(* IEC 61131-3 sources: elnaProjects/ElpcLogic/PomarKc7Changed/FunctionBlocks (part 5) *)

(* ---- OPC_AI_SET.st ---- *)
FUNCTION_BLOCK OPC_AI_SET

VAR_EXTERNAL
	ai : aiConfig;
	AI_Tstali_statora_kanal_1_HL : LREAL;
	AI_Tstali_statora_kanal_1_LL : LREAL;
	AI_Tstali_statora_kanal_1_command : UINT;
	AI_Tstali_statora_kanal_1_newHL : LREAL;
	AI_Tstali_statora_kanal_1_newLL : LREAL;
	AI_Tstali_statora_kanal_1_status : UDINT;
	AI_Tstali_statora_kanal_1_value : LREAL;
	AI_Tstali_statora_kanal_1_HW : LREAL;
	AI_Tstali_statora_kanal_1_newHW : LREAL;
	AI_Tstali_statora_kanal_2_HL : LREAL;
	AI_Tstali_statora_kanal_2_LL : LREAL;
	AI_Tstali_statora_kanal_2_command : UINT;
	AI_Tstali_statora_kanal_2_newHL : LREAL;
	AI_Tstali_statora_kanal_2_newLL : LREAL;
	AI_Tstali_statora_kanal_2_status : UDINT;
	AI_Tstali_statora_kanal_2_value : LREAL;
	AI_Tstali_statora_kanal_2_HW : LREAL;
	AI_Tstali_statora_kanal_2_newHW : LREAL;
	AI_Tstali_statora_kanal_3_HL : LREAL;
	AI_Tstali_statora_kanal_3_LL : LREAL;
	AI_Tstali_statora_kanal_3_command : UINT;
	AI_Tstali_statora_kanal_3_newHL : LREAL;
	AI_Tstali_statora_kanal_3_newLL : LREAL;
	AI_Tstali_statora_kanal_3_status : UDINT;
	AI_Tstali_statora_kanal_3_value : LREAL;
	AI_Tstali_statora_kanal_3_HW : LREAL;
	AI_Tstali_statora_kanal_3_newHW : LREAL;
	AI_Tmedi_statora_kanal_1_HL : LREAL;
	AI_Tmedi_statora_kanal_1_LL : LREAL;
	AI_Tmedi_statora_kanal_1_command : UINT;
	AI_Tmedi_statora_kanal_1_newHL : LREAL;
	AI_Tmedi_statora_kanal_1_newLL : LREAL;
	AI_Tmedi_statora_kanal_1_status : UDINT;
	AI_Tmedi_statora_kanal_1_value : LREAL;
	AI_Tmedi_statora_kanal_1_HW : LREAL;
	AI_Tmedi_statora_kanal_1_newHW : LREAL;
	AI_Tmedi_statora_kanal_2_HL : LREAL;
	AI_Tmedi_statora_kanal_2_LL : LREAL;
	AI_Tmedi_statora_kanal_2_command : UINT;
	AI_Tmedi_statora_kanal_2_newHL : LREAL;
	AI_Tmedi_statora_kanal_2_newLL : LREAL;
	AI_Tmedi_statora_kanal_2_status : UDINT;
	AI_Tmedi_statora_kanal_2_value : LREAL;
	AI_Tmedi_statora_kanal_2_HW : LREAL;
	AI_Tmedi_statora_kanal_2_newHW : LREAL;
	AI_Tmedi_statora_kanal_3_HL : LREAL;
	AI_Tmedi_statora_kanal_3_LL : LREAL;
	AI_Tmedi_statora_kanal_3_command : UINT;
	AI_Tmedi_statora_kanal_3_newHL : LREAL;
	AI_Tmedi_statora_kanal_3_newLL : LREAL;
	AI_Tmedi_statora_kanal_3_status : UDINT;
	AI_Tmedi_statora_kanal_3_value : LREAL;
	AI_Tmedi_statora_kanal_3_HW : LREAL;
	AI_Tmedi_statora_kanal_3_newHW : LREAL;
	AI_Toporno_podshipnika_EDT_1_HL : LREAL;
	AI_Toporno_podshipnika_EDT_1_LL : LREAL;
	AI_Toporno_podshipnika_EDT_1_command : UINT;
	AI_Toporno_podshipnika_EDT_1_newHL : LREAL;
	AI_Toporno_podshipnika_EDT_1_newLL : LREAL;
	AI_Toporno_podshipnika_EDT_1_status : UDINT;
	AI_Toporno_podshipnika_EDT_1_value : LREAL;
	AI_Toporno_podshipnika_EDT_1_HW : LREAL;
	AI_Toporno_podshipnika_EDT_1_newHW : LREAL;
	AI_Toporno_podshipnika_EDT_1_HA : LREAL;
	AI_Toporno_podshipnika_EDT_1_newHA : LREAL;
	AI_Toy_podshipnika_EDT_2_HL : LREAL;
	AI_Toy_podshipnika_EDT_2_LL : LREAL;
	AI_Toy_podshipnika_EDT_2_command : UINT;
	AI_Toy_podshipnika_EDT_2_newHL : LREAL;
	AI_Toy_podshipnika_EDT_2_newLL : LREAL;
	AI_Toy_podshipnika_EDT_2_status : UDINT;
	AI_Toy_podshipnika_EDT_2_value : LREAL;
	AI_Toy_podshipnika_EDT_2_HW : LREAL;
	AI_Toy_podshipnika_EDT_2_newHW : LREAL;
	AI_Toy_podshipnika_EDT_2_HA : LREAL;
	AI_Toy_podshipnika_EDT_2_newHA : LREAL;
	AI_Toy_podshipnika_kol_EDT_3_HL : LREAL;
	AI_Toy_podshipnika_kol_EDT_3_LL : LREAL;
	AI_Toy_podshipnika_kol_EDT_3_command : UINT;
	AI_Toy_podshipnika_kol_EDT_3_newHL : LREAL;
	AI_Toy_podshipnika_kol_EDT_3_newLL : LREAL;
	AI_Toy_podshipnika_kol_EDT_3_status : UDINT;
	AI_Toy_podshipnika_kol_EDT_3_value : LREAL;
	AI_Toy_podshipnika_kol_EDT_3_HW : LREAL;
	AI_Toy_podshipnika_kol_EDT_3_newHW : LREAL;
	AI_Toy_podshipnika_kol_EDT_3_HA : LREAL;
	AI_Toy_podshipnika_kol_EDT_3_newHA : LREAL;
	AI_Toy_podshipnika_kol_EDT_4_HL : LREAL;
	AI_Toy_podshipnika_kol_EDT_4_LL : LREAL;
	AI_Toy_podshipnika_kol_EDT_4_command : UINT;
	AI_Toy_podshipnika_kol_EDT_4_newHL : LREAL;
	AI_Toy_podshipnika_kol_EDT_4_newLL : LREAL;
	AI_Toy_podshipnika_kol_EDT_4_status : UDINT;
	AI_Toy_podshipnika_kol_EDT_4_value : LREAL;
	AI_Toy_podshipnika_kol_EDT_4_HW : LREAL;
	AI_Toy_podshipnika_kol_EDT_4_newHW : LREAL;
	AI_Toy_podshipnika_kol_EDT_4_HA : LREAL;
	AI_Toy_podshipnika_kol_EDT_4_newHA : LREAL;
	AI_Toy_podshipnika_shest_red_EDT_5_HL : LREAL;
	AI_Toy_podshipnika_shest_red_EDT_5_LL : LREAL;
	AI_Toy_podshipnika_shest_red_EDT_5_command : UINT;
	AI_Toy_podshipnika_shest_red_EDT_5_newHL : LREAL;
	AI_Toy_podshipnika_shest_red_EDT_5_newLL : LREAL;
	AI_Toy_podshipnika_shest_red_EDT_5_status : UDINT;
	AI_Toy_podshipnika_shest_red_EDT_5_value : LREAL;
	AI_Toy_podshipnika_shest_red_EDT_5_HW : LREAL;
	AI_Toy_podshipnika_shest_red_EDT_5_newHW : LREAL;
	AI_Toy_podshipnika_shest_red_EDT_5_HA : LREAL;
	AI_Toy_podshipnika_shest_red_EDT_5_newHA : LREAL;
	AI_Ty_podshipnika_red_EDT_6_HL : LREAL;
	AI_Ty_podshipnika_red_EDT_6_LL : LREAL;
	AI_Ty_podshipnika_red_EDT_6_command : UINT;
	AI_Ty_podshipnika_red_EDT_6_newHL : LREAL;
	AI_Ty_podshipnika_red_EDT_6_newLL : LREAL;
	AI_Ty_podshipnika_red_EDT_6_status : UDINT;
	AI_Ty_podshipnika_red_EDT_6_value : LREAL;
	AI_Ty_podshipnika_red_EDT_6_HW : LREAL;
	AI_Ty_podshipnika_red_EDT_6_newHW : LREAL;
	AI_Ty_podshipnika_red_EDT_6_HA : LREAL;
	AI_Ty_podshipnika_red_EDT_6_newHA : LREAL;
	AI_Ty_podshipnika_nagnet_EDT_7_1_HL : LREAL;
	AI_Ty_podshipnika_nagnet_EDT_7_1_LL : LREAL;
	AI_Ty_podshipnika_nagnet_EDT_7_1_command : UINT;
	AI_Ty_podshipnika_nagnet_EDT_7_1_newHL : LREAL;
	AI_Ty_podshipnika_nagnet_EDT_7_1_newLL : LREAL;
	AI_Ty_podshipnika_nagnet_EDT_7_1_status : UDINT;
	AI_Ty_podshipnika_nagnet_EDT_7_1_value : LREAL;
	AI_Ty_podshipnika_nagnet_EDT_7_1_HW : LREAL;
	AI_Ty_podshipnika_nagnet_EDT_7_1_newHW : LREAL;
	AI_Ty_podshipnika_nagnet_EDT_7_1_HA : LREAL;
	AI_Ty_podshipnika_nagnet_EDT_7_1_newHA : LREAL;
	AI_Ty_podshipnika_nagnet_EDT_7_2_HL : LREAL;
	AI_Ty_podshipnika_nagnet_EDT_7_2_LL : LREAL;
	AI_Ty_podshipnika_nagnet_EDT_7_2_command : UINT;
	AI_Ty_podshipnika_nagnet_EDT_7_2_newHL : LREAL;
	AI_Ty_podshipnika_nagnet_EDT_7_2_newLL : LREAL;
	AI_Ty_podshipnika_nagnet_EDT_7_2_status : UDINT;
	AI_Ty_podshipnika_nagnet_EDT_7_2_value : LREAL;
	AI_Ty_podshipnika_nagnet_EDT_7_2_HW : LREAL;
	AI_Ty_podshipnika_nagnet_EDT_7_2_newHW : LREAL;
	AI_Ty_podshipnika_nagnet_EDT_7_2_HA : LREAL;
	AI_Ty_podshipnika_nagnet_EDT_7_2_newHA : LREAL;
	AI_Toy_podshipnika_svobod_konca_EDT_8_1_HL : LREAL;
	AI_Toy_podshipnika_svobod_konca_EDT_8_1_LL : LREAL;
	AI_Toy_podshipnika_svobod_konca_EDT_8_1_command : UINT;
	AI_Toy_podshipnika_svobod_konca_EDT_8_1_newHL : LREAL;
	AI_Toy_podshipnika_svobod_konca_EDT_8_1_newLL : LREAL;
	AI_Toy_podshipnika_svobod_konca_EDT_8_1_status : UDINT;
	AI_Toy_podshipnika_svobod_konca_EDT_8_1_value : LREAL;
	AI_Toy_podshipnika_svobod_konca_EDT_8_1_HW : LREAL;
	AI_Toy_podshipnika_svobod_konca_EDT_8_1_newHW : LREAL;
	AI_Toy_podshipnika_svobod_konca_EDT_8_1_HA : LREAL;
	AI_Toy_podshipnika_svobod_konca_EDT_8_1_newHA : LREAL;
	AI_Toy_podshipnika_svobod_konca_EDT_8_2_HL : LREAL;
	AI_Toy_podshipnika_svobod_konca_EDT_8_2_LL : LREAL;
	AI_Toy_podshipnika_svobod_konca_EDT_8_2_command : UINT;
	AI_Toy_podshipnika_svobod_konca_EDT_8_2_newHL : LREAL;
	AI_Toy_podshipnika_svobod_konca_EDT_8_2_newLL : LREAL;
	AI_Toy_podshipnika_svobod_konca_EDT_8_2_status : UDINT;
	AI_Toy_podshipnika_svobod_konca_EDT_8_2_value : LREAL;
	AI_Toy_podshipnika_svobod_konca_EDT_8_2_HW : LREAL;
	AI_Toy_podshipnika_svobod_konca_EDT_8_2_newHW : LREAL;
	AI_Toy_podshipnika_svobod_konca_EDT_8_2_HA : LREAL;
	AI_Toy_podshipnika_svobod_konca_EDT_8_2_newHA : LREAL;
	AI_Toy_podshipnika_rab_kol_EDT_9_1_HL : LREAL;
	AI_Toy_podshipnika_rab_kol_EDT_9_1_LL : LREAL;
	AI_Toy_podshipnika_rab_kol_EDT_9_1_command : UINT;
	AI_Toy_podshipnika_rab_kol_EDT_9_1_newHL : LREAL;
	AI_Toy_podshipnika_rab_kol_EDT_9_1_newLL : LREAL;
	AI_Toy_podshipnika_rab_kol_EDT_9_1_status : UDINT;
	AI_Toy_podshipnika_rab_kol_EDT_9_1_value : LREAL;
	AI_Toy_podshipnika_rab_kol_EDT_9_1_HW : LREAL;
	AI_Toy_podshipnika_rab_kol_EDT_9_1_newHW : LREAL;
	AI_Toy_podshipnika_rab_kol_EDT_9_1_HA : LREAL;
	AI_Toy_podshipnika_rab_kol_EDT_9_1_newHA : LREAL;
	AI_Toy_podshipnika_rab_kol_EDT_9_2_HL : LREAL;
	AI_Toy_podshipnika_rab_kol_EDT_9_2_LL : LREAL;
	AI_Toy_podshipnika_rab_kol_EDT_9_2_command : UINT;
	AI_Toy_podshipnika_rab_kol_EDT_9_2_newHL : LREAL;
	AI_Toy_podshipnika_rab_kol_EDT_9_2_newLL : LREAL;
	AI_Toy_podshipnika_rab_kol_EDT_9_2_status : UDINT;
	AI_Toy_podshipnika_rab_kol_EDT_9_2_value : LREAL;
	AI_Toy_podshipnika_rab_kol_EDT_9_2_HW : LREAL;
	AI_Toy_podshipnika_rab_kol_EDT_9_2_newHW : LREAL;
	AI_Toy_podshipnika_rab_kol_EDT_9_2_HA : LREAL;
	AI_Toy_podshipnika_rab_kol_EDT_9_2_newHA : LREAL;
	AI_Toy_podshipnika_nerab_kol_EDT_10_1_HL : LREAL;
	AI_Toy_podshipnika_nerab_kol_EDT_10_1_LL : LREAL;
	AI_Toy_podshipnika_nerab_kol_EDT_10_1_command : UINT;
	AI_Toy_podshipnika_nerab_kol_EDT_10_1_newHL : LREAL;
	AI_Toy_podshipnika_nerab_kol_EDT_10_1_newLL : LREAL;
	AI_Toy_podshipnika_nerab_kol_EDT_10_1_status : UDINT;
	AI_Toy_podshipnika_nerab_kol_EDT_10_1_value : LREAL;
	AI_Toy_podshipnika_nerab_kol_EDT_10_1_HW : LREAL;
	AI_Toy_podshipnika_nerab_kol_EDT_10_1_newHW : LREAL;
	AI_Toy_podshipnika_nerab_kol_EDT_10_1_HA : LREAL;
	AI_Toy_podshipnika_nerab_kol_EDT_10_1_newHA : LREAL;
	AI_Toy_podshipnika_nerab_kol_EDT_10_2_HL : LREAL;
	AI_Toy_podshipnika_nerab_kol_EDT_10_2_LL : LREAL;
	AI_Toy_podshipnika_nerab_kol_EDT_10_2_command : UINT;
	AI_Toy_podshipnika_nerab_kol_EDT_10_2_newHL : LREAL;
	AI_Toy_podshipnika_nerab_kol_EDT_10_2_newLL : LREAL;
	AI_Toy_podshipnika_nerab_kol_EDT_10_2_status : UDINT;
	AI_Toy_podshipnika_nerab_kol_EDT_10_2_value : LREAL;
	AI_Toy_podshipnika_nerab_kol_EDT_10_2_HW : LREAL;
	AI_Toy_podshipnika_nerab_kol_EDT_10_2_newHW : LREAL;
	AI_Toy_podshipnika_nerab_kol_EDT_10_2_HA : LREAL;
	AI_Toy_podshipnika_nerab_kol_EDT_10_2_newHA : LREAL;
	AI_Tholodnogo_vozduha_ED_kanal_1_HL : LREAL;
	AI_Tholodnogo_vozduha_ED_kanal_1_LL : LREAL;
	AI_Tholodnogo_vozduha_ED_kanal_1_command : UINT;
	AI_Tholodnogo_vozduha_ED_kanal_1_newHL : LREAL;
	AI_Tholodnogo_vozduha_ED_kanal_1_newLL : LREAL;
	AI_Tholodnogo_vozduha_ED_kanal_1_status : UDINT;
	AI_Tholodnogo_vozduha_ED_kanal_1_value : LREAL;
	AI_Tholodnogo_vozduha_ED_kanal_1_HW : LREAL;
	AI_Tholodnogo_vozduha_ED_kanal_1_newHW : LREAL;
	AI_Tholodnogo_vozduha_ED_kanal_2_HL : LREAL;
	AI_Tholodnogo_vozduha_ED_kanal_2_LL : LREAL;
	AI_Tholodnogo_vozduha_ED_kanal_2_command : UINT;
	AI_Tholodnogo_vozduha_ED_kanal_2_newHL : LREAL;
	AI_Tholodnogo_vozduha_ED_kanal_2_newLL : LREAL;
	AI_Tholodnogo_vozduha_ED_kanal_2_status : UDINT;
	AI_Tholodnogo_vozduha_ED_kanal_2_value : LREAL;
	AI_Tholodnogo_vozduha_ED_kanal_2_HW : LREAL;
	AI_Tholodnogo_vozduha_ED_kanal_2_newHW : LREAL;
	AI_Tgorjachego_vozduha_ED_kanal_1_HL : LREAL;
	AI_Tgorjachego_vozduha_ED_kanal_1_LL : LREAL;
	AI_Tgorjachego_vozduha_ED_kanal_1_command : UINT;
	AI_Tgorjachego_vozduha_ED_kanal_1_newHL : LREAL;
	AI_Tgorjachego_vozduha_ED_kanal_1_newLL : LREAL;
	AI_Tgorjachego_vozduha_ED_kanal_1_status : UDINT;
	AI_Tgorjachego_vozduha_ED_kanal_1_value : LREAL;
	AI_Tgorjachego_vozduha_ED_kanal_1_HW : LREAL;
	AI_Tgorjachego_vozduha_ED_kanal_1_newHW : LREAL;
	AI_Tgorjachego_vozduha_ED_kanal_2_HL : LREAL;
	AI_Tgorjachego_vozduha_ED_kanal_2_LL : LREAL;
	AI_Tgorjachego_vozduha_ED_kanal_2_command : UINT;
	AI_Tgorjachego_vozduha_ED_kanal_2_newHL : LREAL;
	AI_Tgorjachego_vozduha_ED_kanal_2_newLL : LREAL;
	AI_Tgorjachego_vozduha_ED_kanal_2_status : UDINT;
	AI_Tgorjachego_vozduha_ED_kanal_2_value : LREAL;
	AI_Tgorjachego_vozduha_ED_kanal_2_HW : LREAL;
	AI_Tgorjachego_vozduha_ED_kanal_2_newHW : LREAL;
	AI_Tnarujnogo_vozduha_HL : LREAL;
	AI_Tnarujnogo_vozduha_LL : LREAL;
	AI_Tnarujnogo_vozduha_command : UINT;
	AI_Tnarujnogo_vozduha_newHL : LREAL;
	AI_Tnarujnogo_vozduha_newLL : LREAL;
	AI_Tnarujnogo_vozduha_status : UDINT;
	AI_Tnarujnogo_vozduha_value : LREAL;
	AI_Tnarujnogo_vozduha_HW : LREAL;
	AI_Tnarujnogo_vozduha_newHW : LREAL;
	AI_Tgaza_na_vhode_H_HL : LREAL;
	AI_Tgaza_na_vhode_H_LL : LREAL;
	AI_Tgaza_na_vhode_H_command : UINT;
	AI_Tgaza_na_vhode_H_newHL : LREAL;
	AI_Tgaza_na_vhode_H_newLL : LREAL;
	AI_Tgaza_na_vhode_H_status : UDINT;
	AI_Tgaza_na_vhode_H_value : LREAL;
	AI_Tgaza_na_vhode_H_HW : LREAL;
	AI_Tgaza_na_vhode_H_newHW : LREAL;
	AI_Tgaza_na_vyhode_H_HL : LREAL;
	AI_Tgaza_na_vyhode_H_LL : LREAL;
	AI_Tgaza_na_vyhode_H_command : UINT;
	AI_Tgaza_na_vyhode_H_newHL : LREAL;
	AI_Tgaza_na_vyhode_H_newLL : LREAL;
	AI_Tgaza_na_vyhode_H_status : UDINT;
	AI_Tgaza_na_vyhode_H_value : LREAL;
	AI_Tgaza_na_vyhode_H_HW : LREAL;
	AI_Tgaza_na_vyhode_H_newHW : LREAL;
	AI_Tgaza_na_vyhode_H_HA : LREAL;
	AI_Tgaza_na_vyhode_H_newHA : LREAL;
	AI_Tmasla_do_AVOM_HL : LREAL;
	AI_Tmasla_do_AVOM_LL : LREAL;
	AI_Tmasla_do_AVOM_command : UINT;
	AI_Tmasla_do_AVOM_newHL : LREAL;
	AI_Tmasla_do_AVOM_newLL : LREAL;
	AI_Tmasla_do_AVOM_status : UDINT;
	AI_Tmasla_do_AVOM_value : LREAL;
	AI_Tmasla_do_AVOM_HW : LREAL;
	AI_Tmasla_do_AVOM_newHW : LREAL;
	AI_Tmasla_posle_AVOM_HL : LREAL;
	AI_Tmasla_posle_AVOM_LL : LREAL;
	AI_Tmasla_posle_AVOM_command : UINT;
	AI_Tmasla_posle_AVOM_newHL : LREAL;
	AI_Tmasla_posle_AVOM_newLL : LREAL;
	AI_Tmasla_posle_AVOM_status : UDINT;
	AI_Tmasla_posle_AVOM_value : LREAL;
	AI_Tmasla_posle_AVOM_HW : LREAL;
	AI_Tmasla_posle_AVOM_newHW : LREAL;
	AI_Tmasla_MB_HL : LREAL;
	AI_Tmasla_MB_LL : LREAL;
	AI_Tmasla_MB_command : UINT;
	AI_Tmasla_MB_newHL : LREAL;
	AI_Tmasla_MB_newLL : LREAL;
	AI_Tmasla_MB_status : UDINT;
	AI_Tmasla_MB_value : LREAL;
	AI_Tmasla_MB_HW : LREAL;
	AI_Tmasla_MB_newHW : LREAL;
	AI_Tmasla_MB_TEN_HL : LREAL;
	AI_Tmasla_MB_TEN_LL : LREAL;
	AI_Tmasla_MB_TEN_command : UINT;
	AI_Tmasla_MB_TEN_newHL : LREAL;
	AI_Tmasla_MB_TEN_newLL : LREAL;
	AI_Tmasla_MB_TEN_status : UDINT;
	AI_Tmasla_MB_TEN_value : LREAL;
	AI_Tmasla_MB_TEN_HW : LREAL;
	AI_Tmasla_MB_TEN_newHW : LREAL;
	AI_Tshu_HL : LREAL;
	AI_Tshu_LL : LREAL;
	AI_Tshu_command : UINT;
	AI_Tshu_newHL : LREAL;
	AI_Tshu_newLL : LREAL;
	AI_Tshu_status : UDINT;
	AI_Tshu_value : LREAL;
	AI_Pmaslo_sm_nizkoe_HL : LREAL;
	AI_Pmaslo_sm_nizkoe_LL : LREAL;
	AI_Pmaslo_sm_nizkoe_command : UINT;
	AI_Pmaslo_sm_nizkoe_newHL : LREAL;
	AI_Pmaslo_sm_nizkoe_newLL : LREAL;
	AI_Pmaslo_sm_nizkoe_status : UDINT;
	AI_Pmaslo_sm_nizkoe_value : LREAL;
	AI_Pmaslo_sm_nizkoe_LW : LREAL;
	AI_Pmaslo_sm_nizkoe_newLW : LREAL;
	AI_Pmaslo_sm_nizkoe_LA : LREAL;
	AI_Pmaslo_sm_nizkoe_newLA : LREAL;
	AI_Pmaslo_sm_vysokoe_HL : LREAL;
	AI_Pmaslo_sm_vysokoe_LL : LREAL;
	AI_Pmaslo_sm_vysokoe_command : UINT;
	AI_Pmaslo_sm_vysokoe_newHL : LREAL;
	AI_Pmaslo_sm_vysokoe_newLL : LREAL;
	AI_Pmaslo_sm_vysokoe_status : UDINT;
	AI_Pmaslo_sm_vysokoe_value : LREAL;
	AI_Pmaslo_sm_vysokoe_LW : LREAL;
	AI_Pmaslo_sm_vysokoe_newLW : LREAL;
	AI_Pmaslo_sm_vysokoe_LA : LREAL;
	AI_Pmaslo_sm_vysokoe_newLA : LREAL;
	AI_Pmasla_posle_GNS_HL : LREAL;
	AI_Pmasla_posle_GNS_LL : LREAL;
	AI_Pmasla_posle_GNS_command : UINT;
	AI_Pmasla_posle_GNS_newHL : LREAL;
	AI_Pmasla_posle_GNS_newLL : LREAL;
	AI_Pmasla_posle_GNS_status : UDINT;
	AI_Pmasla_posle_GNS_value : LREAL;
	AI_Pmasla_posle_GNS_HW : LREAL;
	AI_Pmasla_posle_GNS_newHW : LREAL;
	AI_Pmasla_posle_GNS_LW : LREAL;
	AI_Pmasla_posle_GNS_newLW : LREAL;
	AI_Pmasla_posle_NU_HL : LREAL;
	AI_Pmasla_posle_NU_LL : LREAL;
	AI_Pmasla_posle_NU_command : UINT;
	AI_Pmasla_posle_NU_newHL : LREAL;
	AI_Pmasla_posle_NU_newLL : LREAL;
	AI_Pmasla_posle_NU_status : UDINT;
	AI_Pmasla_posle_NU_value : LREAL;
	AI_Pmasla_posle_NU_LW : LREAL;
	AI_Pmasla_posle_NU_newLW : LREAL;
	AI_Pgaza_na_vhode_nagnetatelia_HL : LREAL;
	AI_Pgaza_na_vhode_nagnetatelia_LL : LREAL;
	AI_Pgaza_na_vhode_nagnetatelia_command : UINT;
	AI_Pgaza_na_vhode_nagnetatelia_newHL : LREAL;
	AI_Pgaza_na_vhode_nagnetatelia_newLL : LREAL;
	AI_Pgaza_na_vhode_nagnetatelia_status : UDINT;
	AI_Pgaza_na_vhode_nagnetatelia_value : LREAL;
	AI_Pgaza_na_vhode_nagnetatelia_LW : LREAL;
	AI_Pgaza_na_vhode_nagnetatelia_newLW : LREAL;
	AI_Pgaza_na_vyhode_nagnetatelia_HL : LREAL;
	AI_Pgaza_na_vyhode_nagnetatelia_LL : LREAL;
	AI_Pgaza_na_vyhode_nagnetatelia_command : UINT;
	AI_Pgaza_na_vyhode_nagnetatelia_newHL : LREAL;
	AI_Pgaza_na_vyhode_nagnetatelia_newLL : LREAL;
	AI_Pgaza_na_vyhode_nagnetatelia_status : UDINT;
	AI_Pgaza_na_vyhode_nagnetatelia_value : LREAL;
	AI_Pgaza_na_vyhode_nagnetatelia_LW : LREAL;
	AI_Pgaza_na_vyhode_nagnetatelia_newLW : LREAL;
	AI_Pgaza_na_vyhode_nagnetatelia_HA : LREAL;
	AI_Pgaza_na_vyhode_nagnetatelia_newHA : LREAL;
	AI_Pimpuls_gaz_HL : LREAL;
	AI_Pimpuls_gaz_LL : LREAL;
	AI_Pimpuls_gaz_command : UINT;
	AI_Pimpuls_gaz_newHL : LREAL;
	AI_Pimpuls_gaz_newLL : LREAL;
	AI_Pimpuls_gaz_status : UDINT;
	AI_Pimpuls_gaz_value : LREAL;
	AI_Pimpuls_gaz_LW : LREAL;
	AI_Pimpuls_gaz_newLW : LREAL;
	AI_dPgaza_na_maslo_filtre_HL : LREAL;
	AI_dPgaza_na_maslo_filtre_LL : LREAL;
	AI_dPgaza_na_maslo_filtre_command : UINT;
	AI_dPgaza_na_maslo_filtre_newHL : LREAL;
	AI_dPgaza_na_maslo_filtre_newLL : LREAL;
	AI_dPgaza_na_maslo_filtre_status : UDINT;
	AI_dPgaza_na_maslo_filtre_value : LREAL;
	AI_dPgaza_na_maslo_filtre_HW : LREAL;
	AI_dPgaza_na_maslo_filtre_newHW : LREAL;
	AI_dPgaza_na_konfuzore_HL : LREAL;
	AI_dPgaza_na_konfuzore_LL : LREAL;
	AI_dPgaza_na_konfuzore_command : UINT;
	AI_dPgaza_na_konfuzore_newHL : LREAL;
	AI_dPgaza_na_konfuzore_newLL : LREAL;
	AI_dPgaza_na_konfuzore_status : UDINT;
	AI_dPgaza_na_konfuzore_value : LREAL;
	AI_dPgaza_na_konfuzore_LW : LREAL;
	AI_dPgaza_na_konfuzore_newLW : LREAL;
	AI_dPmaslo_gaz_HL : LREAL;
	AI_dPmaslo_gaz_LL : LREAL;
	AI_dPmaslo_gaz_command : UINT;
	AI_dPmaslo_gaz_newHL : LREAL;
	AI_dPmaslo_gaz_newLL : LREAL;
	AI_dPmaslo_gaz_status : UDINT;
	AI_dPmaslo_gaz_value : LREAL;
	AI_dPmaslo_gaz_LW : LREAL;
	AI_dPmaslo_gaz_newLW : LREAL;
	AI_dPmaslo_gaz_LA : LREAL;
	AI_dPmaslo_gaz_newLA : LREAL;
	AI_Os_sdvig_nagnetatelja_plus_HL : LREAL;
	AI_Os_sdvig_nagnetatelja_plus_LL : LREAL;
	AI_Os_sdvig_nagnetatelja_plus_command : UINT;
	AI_Os_sdvig_nagnetatelja_plus_newHL : LREAL;
	AI_Os_sdvig_nagnetatelja_plus_newLL : LREAL;
	AI_Os_sdvig_nagnetatelja_plus_status : UDINT;
	AI_Os_sdvig_nagnetatelja_plus_value : LREAL;
	AI_Os_sdvig_nagnetatelja_plus_HW : LREAL;
	AI_Os_sdvig_nagnetatelja_plus_newHW : LREAL;
	AI_Os_sdvig_nagnetatelja_plus_HA : LREAL;
	AI_Os_sdvig_nagnetatelja_plus_newHA : LREAL;
	AI_Os_sdvig_nagnetatelja_minus_HL : LREAL;
	AI_Os_sdvig_nagnetatelja_minus_LL : LREAL;
	AI_Os_sdvig_nagnetatelja_minus_command : UINT;
	AI_Os_sdvig_nagnetatelja_minus_newHL : LREAL;
	AI_Os_sdvig_nagnetatelja_minus_newLL : LREAL;
	AI_Os_sdvig_nagnetatelja_minus_status : UDINT;
	AI_Os_sdvig_nagnetatelja_minus_value : LREAL;
	AI_Os_sdvig_nagnetatelja_minus_LW : LREAL;
	AI_Os_sdvig_nagnetatelja_minus_newLW : LREAL;
	AI_Os_sdvig_nagnetatelja_minus_LA : LREAL;
	AI_Os_sdvig_nagnetatelja_minus_newLA : LREAL;
	AI_Yroven_masla_MB_HL : LREAL;
	AI_Yroven_masla_MB_LL : LREAL;
	AI_Yroven_masla_MB_command : UINT;
	AI_Yroven_masla_MB_newHL : LREAL;
	AI_Yroven_masla_MB_newLL : LREAL;
	AI_Yroven_masla_MB_status : UDINT;
	AI_Yroven_masla_MB_value : LREAL;
	AI_Yroven_masla_MB_LW : LREAL;
	AI_Yroven_masla_MB_newLW : LREAL;
	AI_Kontrol_per_220V_HL : LREAL;
	AI_Kontrol_per_220V_LL : LREAL;
	AI_Kontrol_per_220V_command : UINT;
	AI_Kontrol_per_220V_newHL : LREAL;
	AI_Kontrol_per_220V_newLL : LREAL;
	AI_Kontrol_per_220V_status : UDINT;
	AI_Kontrol_per_220V_value : LREAL;
	AI_Kontrol_per_220V_HW : LREAL;
	AI_Kontrol_per_220V_newHW : LREAL;
	AI_Kontrol_per_220V_LW : LREAL;
	AI_Kontrol_per_220V_newLW : LREAL;
	AI_Kontrol_post_220V_HL : LREAL;
	AI_Kontrol_post_220V_LL : LREAL;
	AI_Kontrol_post_220V_command : UINT;
	AI_Kontrol_post_220V_newHL : LREAL;
	AI_Kontrol_post_220V_newLL : LREAL;
	AI_Kontrol_post_220V_status : UDINT;
	AI_Kontrol_post_220V_value : LREAL;
	AI_Kontrol_post_220V_HW : LREAL;
	AI_Kontrol_post_220V_newHW : LREAL;
	AI_Kontrol_post_220V_LW : LREAL;
	AI_Kontrol_post_220V_newLW : LREAL;
	AI_Tok_statora_HL : LREAL;
	AI_Tok_statora_LL : LREAL;
	AI_Tok_statora_command : UINT;
	AI_Tok_statora_newHL : LREAL;
	AI_Tok_statora_newLL : LREAL;
	AI_Tok_statora_status : UDINT;
	AI_Tok_statora_value : LREAL;
	AI_Tok_statora_LW : LREAL;
	AI_Tok_statora_newLW : LREAL;
	AI_Vibro_skorost_OPED_T1_HL : LREAL;
	AI_Vibro_skorost_OPED_T1_LL : LREAL;
	AI_Vibro_skorost_OPED_T1_command : UINT;
	AI_Vibro_skorost_OPED_T1_newHL : LREAL;
	AI_Vibro_skorost_OPED_T1_newLL : LREAL;
	AI_Vibro_skorost_OPED_T1_status : UDINT;
	AI_Vibro_skorost_OPED_T1_value : LREAL;
	AI_Vibro_skorost_OPED_T1_HW : LREAL;
	AI_Vibro_skorost_OPED_T1_newHW : LREAL;
	AI_Vibro_skorost_OPED_T1_HA : LREAL;
	AI_Vibro_skorost_OPED_T1_newHA : LREAL;
	AI_Vibro_skorost_OYPED_T2_HL : LREAL;
	AI_Vibro_skorost_OYPED_T2_LL : LREAL;
	AI_Vibro_skorost_OYPED_T2_command : UINT;
	AI_Vibro_skorost_OYPED_T2_newHL : LREAL;
	AI_Vibro_skorost_OYPED_T2_newLL : LREAL;
	AI_Vibro_skorost_OYPED_T2_status : UDINT;
	AI_Vibro_skorost_OYPED_T2_value : LREAL;
	AI_Vibro_skorost_OYPED_T2_HW : LREAL;
	AI_Vibro_skorost_OYPED_T2_newHW : LREAL;
	AI_Vibro_skorost_OYPED_T2_HA : LREAL;
	AI_Vibro_skorost_OYPED_T2_newHA : LREAL;
	AI_Vibro_skorost_OYP_kolesa_ED_T3_HL : LREAL;
	AI_Vibro_skorost_OYP_kolesa_ED_T3_LL : LREAL;
	AI_Vibro_skorost_OYP_kolesa_ED_T3_command : UINT;
	AI_Vibro_skorost_OYP_kolesa_ED_T3_newHL : LREAL;
	AI_Vibro_skorost_OYP_kolesa_ED_T3_newLL : LREAL;
	AI_Vibro_skorost_OYP_kolesa_ED_T3_status : UDINT;
	AI_Vibro_skorost_OYP_kolesa_ED_T3_value : LREAL;
	AI_Vibro_skorost_OYP_kolesa_ED_T3_HW : LREAL;
	AI_Vibro_skorost_OYP_kolesa_ED_T3_newHW : LREAL;
	AI_Vibro_skorost_OYP_kolesa_ED_T3_HA : LREAL;
	AI_Vibro_skorost_OYP_kolesa_ED_T3_newHA : LREAL;
	AI_Vibro_skorost_OP_kolesa_RH_T4_HL : LREAL;
	AI_Vibro_skorost_OP_kolesa_RH_T4_LL : LREAL;
	AI_Vibro_skorost_OP_kolesa_RH_T4_command : UINT;
	AI_Vibro_skorost_OP_kolesa_RH_T4_newHL : LREAL;
	AI_Vibro_skorost_OP_kolesa_RH_T4_newLL : LREAL;
	AI_Vibro_skorost_OP_kolesa_RH_T4_status : UDINT;
	AI_Vibro_skorost_OP_kolesa_RH_T4_value : LREAL;
	AI_Vibro_skorost_OP_kolesa_RH_T4_HW : LREAL;
	AI_Vibro_skorost_OP_kolesa_RH_T4_newHW : LREAL;
	AI_Vibro_skorost_OP_kolesa_RH_T4_HA : LREAL;
	AI_Vibro_skorost_OP_kolesa_RH_T4_newHA : LREAL;
	AI_Vibro_skorost_OP_shesterni_RED_T5_HL : LREAL;
	AI_Vibro_skorost_OP_shesterni_RED_T5_LL : LREAL;
	AI_Vibro_skorost_OP_shesterni_RED_T5_command : UINT;
	AI_Vibro_skorost_OP_shesterni_RED_T5_newHL : LREAL;
	AI_Vibro_skorost_OP_shesterni_RED_T5_newLL : LREAL;
	AI_Vibro_skorost_OP_shesterni_RED_T5_status : UDINT;
	AI_Vibro_skorost_OP_shesterni_RED_T5_value : LREAL;
	AI_Vibro_skorost_OP_shesterni_RED_T5_HW : LREAL;
	AI_Vibro_skorost_OP_shesterni_RED_T5_newHW : LREAL;
	AI_Vibro_skorost_OP_shesterni_RED_T5_HA : LREAL;
	AI_Vibro_skorost_OP_shesterni_RED_T5_newHA : LREAL;
	AI_Vibro_skorost_OP_shesterni_RED_T6_HL : LREAL;
	AI_Vibro_skorost_OP_shesterni_RED_T6_LL : LREAL;
	AI_Vibro_skorost_OP_shesterni_RED_T6_command : UINT;
	AI_Vibro_skorost_OP_shesterni_RED_T6_newHL : LREAL;
	AI_Vibro_skorost_OP_shesterni_RED_T6_newLL : LREAL;
	AI_Vibro_skorost_OP_shesterni_RED_T6_status : UDINT;
	AI_Vibro_skorost_OP_shesterni_RED_T6_value : LREAL;
	AI_Vibro_skorost_OP_shesterni_RED_T6_HW : LREAL;
	AI_Vibro_skorost_OP_shesterni_RED_T6_newHW : LREAL;
	AI_Vibro_skorost_OP_shesterni_RED_T6_HA : LREAL;
	AI_Vibro_skorost_OP_shesterni_RED_T6_newHA : LREAL;
END_VAR

AI_Tstali_statora_kanal_1_HL := ai.Tstali_statora_kanal_1.HL;
AI_Tstali_statora_kanal_1_LL := ai.Tstali_statora_kanal_1.LL;
AI_Tstali_statora_kanal_1_status := DWORD_TO_UDINT(ai.Tstali_statora_kanal_1.status);
AI_Tstali_statora_kanal_1_value := ai.Tstali_statora_kanal_1.value;
AI_Tstali_statora_kanal_1_HW := ai.Tstali_statora_kanal_1.HW;

AI_Tstali_statora_kanal_2_HL := ai.Tstali_statora_kanal_2.HL;
AI_Tstali_statora_kanal_2_LL := ai.Tstali_statora_kanal_2.LL;
AI_Tstali_statora_kanal_2_status := DWORD_TO_UDINT(ai.Tstali_statora_kanal_2.status);
AI_Tstali_statora_kanal_2_value := ai.Tstali_statora_kanal_2.value;
AI_Tstali_statora_kanal_2_HW := ai.Tstali_statora_kanal_2.HW;

AI_Tstali_statora_kanal_3_HL := ai.Tstali_statora_kanal_3.HL;
AI_Tstali_statora_kanal_3_LL := ai.Tstali_statora_kanal_3.LL;
AI_Tstali_statora_kanal_3_status := DWORD_TO_UDINT(ai.Tstali_statora_kanal_3.status);
AI_Tstali_statora_kanal_3_value := ai.Tstali_statora_kanal_3.value;
AI_Tstali_statora_kanal_3_HW := ai.Tstali_statora_kanal_3.HW;

AI_Tmedi_statora_kanal_1_HL := ai.Tmedi_statora_kanal_1.HL;
AI_Tmedi_statora_kanal_1_LL := ai.Tmedi_statora_kanal_1.LL;
AI_Tmedi_statora_kanal_1_status := DWORD_TO_UDINT(ai.Tmedi_statora_kanal_1.status);
AI_Tmedi_statora_kanal_1_value := ai.Tmedi_statora_kanal_1.value;
AI_Tmedi_statora_kanal_1_HW := ai.Tmedi_statora_kanal_1.HW;

AI_Tmedi_statora_kanal_2_HL := ai.Tmedi_statora_kanal_2.HL;
AI_Tmedi_statora_kanal_2_LL := ai.Tmedi_statora_kanal_2.LL;
AI_Tmedi_statora_kanal_2_status := DWORD_TO_UDINT(ai.Tmedi_statora_kanal_2.status);
AI_Tmedi_statora_kanal_2_value := ai.Tmedi_statora_kanal_2.value;
AI_Tmedi_statora_kanal_2_HW := ai.Tmedi_statora_kanal_2.HW;

AI_Tmedi_statora_kanal_3_HL := ai.Tmedi_statora_kanal_3.HL;
AI_Tmedi_statora_kanal_3_LL := ai.Tmedi_statora_kanal_3.LL;
AI_Tmedi_statora_kanal_3_status := DWORD_TO_UDINT(ai.Tmedi_statora_kanal_3.status);
AI_Tmedi_statora_kanal_3_value := ai.Tmedi_statora_kanal_3.value;
AI_Tmedi_statora_kanal_3_HW := ai.Tmedi_statora_kanal_3.HW;

AI_Toporno_podshipnika_EDT_1_HL := ai.Toporno_podshipnika_EDT_1.HL;
AI_Toporno_podshipnika_EDT_1_LL := ai.Toporno_podshipnika_EDT_1.LL;
AI_Toporno_podshipnika_EDT_1_status := DWORD_TO_UDINT(ai.Toporno_podshipnika_EDT_1.status);
AI_Toporno_podshipnika_EDT_1_value := ai.Toporno_podshipnika_EDT_1.value;
AI_Toporno_podshipnika_EDT_1_HW := ai.Toporno_podshipnika_EDT_1.HW;
AI_Toporno_podshipnika_EDT_1_HA := ai.Toporno_podshipnika_EDT_1.HA;

AI_Toy_podshipnika_EDT_2_HL := ai.Toy_podshipnika_EDT_2.HL;
AI_Toy_podshipnika_EDT_2_LL := ai.Toy_podshipnika_EDT_2.LL;
AI_Toy_podshipnika_EDT_2_status := DWORD_TO_UDINT(ai.Toy_podshipnika_EDT_2.status);
AI_Toy_podshipnika_EDT_2_value := ai.Toy_podshipnika_EDT_2.value;
AI_Toy_podshipnika_EDT_2_HW := ai.Toy_podshipnika_EDT_2.HW;
AI_Toy_podshipnika_EDT_2_HA := ai.Toy_podshipnika_EDT_2.HA;

AI_Toy_podshipnika_kol_EDT_3_HL := ai.Toy_podshipnika_kol_EDT_3.HL;
AI_Toy_podshipnika_kol_EDT_3_LL := ai.Toy_podshipnika_kol_EDT_3.LL;
AI_Toy_podshipnika_kol_EDT_3_status := DWORD_TO_UDINT(ai.Toy_podshipnika_kol_EDT_3.status);
AI_Toy_podshipnika_kol_EDT_3_value := ai.Toy_podshipnika_kol_EDT_3.value;
AI_Toy_podshipnika_kol_EDT_3_HW := ai.Toy_podshipnika_kol_EDT_3.HW;
AI_Toy_podshipnika_kol_EDT_3_HA := ai.Toy_podshipnika_kol_EDT_3.HA;

AI_Toy_podshipnika_kol_EDT_4_HL := ai.Toy_podshipnika_kol_EDT_4.HL;
AI_Toy_podshipnika_kol_EDT_4_LL := ai.Toy_podshipnika_kol_EDT_4.LL;
AI_Toy_podshipnika_kol_EDT_4_status := DWORD_TO_UDINT(ai.Toy_podshipnika_kol_EDT_4.status);
AI_Toy_podshipnika_kol_EDT_4_value := ai.Toy_podshipnika_kol_EDT_4.value;
AI_Toy_podshipnika_kol_EDT_4_HW := ai.Toy_podshipnika_kol_EDT_4.HW;
AI_Toy_podshipnika_kol_EDT_4_HA := ai.Toy_podshipnika_kol_EDT_4.HA;

AI_Toy_podshipnika_shest_red_EDT_5_HL := ai.Toy_podshipnika_shest_red_EDT_5.HL;
AI_Toy_podshipnika_shest_red_EDT_5_LL := ai.Toy_podshipnika_shest_red_EDT_5.LL;
AI_Toy_podshipnika_shest_red_EDT_5_status := DWORD_TO_UDINT(ai.Toy_podshipnika_shest_red_EDT_5.status);
AI_Toy_podshipnika_shest_red_EDT_5_value := ai.Toy_podshipnika_shest_red_EDT_5.value;
AI_Toy_podshipnika_shest_red_EDT_5_HW := ai.Toy_podshipnika_shest_red_EDT_5.HW;
AI_Toy_podshipnika_shest_red_EDT_5_HA := ai.Toy_podshipnika_shest_red_EDT_5.HA;

AI_Ty_podshipnika_red_EDT_6_HL := ai.Ty_podshipnika_red_EDT_6.HL;
AI_Ty_podshipnika_red_EDT_6_LL := ai.Ty_podshipnika_red_EDT_6.LL;
AI_Ty_podshipnika_red_EDT_6_status := DWORD_TO_UDINT(ai.Ty_podshipnika_red_EDT_6.status);
AI_Ty_podshipnika_red_EDT_6_value := ai.Ty_podshipnika_red_EDT_6.value;
AI_Ty_podshipnika_red_EDT_6_HW := ai.Ty_podshipnika_red_EDT_6.HW;
AI_Ty_podshipnika_red_EDT_6_HA := ai.Ty_podshipnika_red_EDT_6.HA;

AI_Ty_podshipnika_nagnet_EDT_7_1_HL := ai.Ty_podshipnika_nagnet_EDT_7_1.HL;
AI_Ty_podshipnika_nagnet_EDT_7_1_LL := ai.Ty_podshipnika_nagnet_EDT_7_1.LL;
AI_Ty_podshipnika_nagnet_EDT_7_1_status := DWORD_TO_UDINT(ai.Ty_podshipnika_nagnet_EDT_7_1.status);
AI_Ty_podshipnika_nagnet_EDT_7_1_value := ai.Ty_podshipnika_nagnet_EDT_7_1.value;
AI_Ty_podshipnika_nagnet_EDT_7_1_HW := ai.Ty_podshipnika_nagnet_EDT_7_1.HW;
AI_Ty_podshipnika_nagnet_EDT_7_1_HA := ai.Ty_podshipnika_nagnet_EDT_7_1.HA;

AI_Ty_podshipnika_nagnet_EDT_7_2_HL := ai.Ty_podshipnika_nagnet_EDT_7_2.HL;
AI_Ty_podshipnika_nagnet_EDT_7_2_LL := ai.Ty_podshipnika_nagnet_EDT_7_2.LL;
AI_Ty_podshipnika_nagnet_EDT_7_2_status := DWORD_TO_UDINT(ai.Ty_podshipnika_nagnet_EDT_7_2.status);
AI_Ty_podshipnika_nagnet_EDT_7_2_value := ai.Ty_podshipnika_nagnet_EDT_7_2.value;
AI_Ty_podshipnika_nagnet_EDT_7_2_HW := ai.Ty_podshipnika_nagnet_EDT_7_2.HW;
AI_Ty_podshipnika_nagnet_EDT_7_2_HA := ai.Ty_podshipnika_nagnet_EDT_7_2.HA;

AI_Toy_podshipnika_svobod_konca_EDT_8_1_HL := ai.Toy_podshipnika_svobod_konca_EDT_8_1.HL;
AI_Toy_podshipnika_svobod_konca_EDT_8_1_LL := ai.Toy_podshipnika_svobod_konca_EDT_8_1.LL;
AI_Toy_podshipnika_svobod_konca_EDT_8_1_status := DWORD_TO_UDINT(ai.Toy_podshipnika_svobod_konca_EDT_8_1.status);
AI_Toy_podshipnika_svobod_konca_EDT_8_1_value := ai.Toy_podshipnika_svobod_konca_EDT_8_1.value;
AI_Toy_podshipnika_svobod_konca_EDT_8_1_HW := ai.Toy_podshipnika_svobod_konca_EDT_8_1.HW;
AI_Toy_podshipnika_svobod_konca_EDT_8_1_HA := ai.Toy_podshipnika_svobod_konca_EDT_8_1.HA;

AI_Toy_podshipnika_svobod_konca_EDT_8_2_HL := ai.Toy_podshipnika_svobod_konca_EDT_8_2.HL;
AI_Toy_podshipnika_svobod_konca_EDT_8_2_LL := ai.Toy_podshipnika_svobod_konca_EDT_8_2.LL;
AI_Toy_podshipnika_svobod_konca_EDT_8_2_status := DWORD_TO_UDINT(ai.Toy_podshipnika_svobod_konca_EDT_8_2.status);
AI_Toy_podshipnika_svobod_konca_EDT_8_2_value := ai.Toy_podshipnika_svobod_konca_EDT_8_2.value;
AI_Toy_podshipnika_svobod_konca_EDT_8_2_HW := ai.Toy_podshipnika_svobod_konca_EDT_8_2.HW;
AI_Toy_podshipnika_svobod_konca_EDT_8_2_HA := ai.Toy_podshipnika_svobod_konca_EDT_8_2.HA;

AI_Toy_podshipnika_rab_kol_EDT_9_1_HL := ai.Toy_podshipnika_rab_kol_EDT_9_1.HL;
AI_Toy_podshipnika_rab_kol_EDT_9_1_LL := ai.Toy_podshipnika_rab_kol_EDT_9_1.LL;
AI_Toy_podshipnika_rab_kol_EDT_9_1_status := DWORD_TO_UDINT(ai.Toy_podshipnika_rab_kol_EDT_9_1.status);
AI_Toy_podshipnika_rab_kol_EDT_9_1_value := ai.Toy_podshipnika_rab_kol_EDT_9_1.value;
AI_Toy_podshipnika_rab_kol_EDT_9_1_HW := ai.Toy_podshipnika_rab_kol_EDT_9_1.HW;
AI_Toy_podshipnika_rab_kol_EDT_9_1_HA := ai.Toy_podshipnika_rab_kol_EDT_9_1.HA;

AI_Toy_podshipnika_rab_kol_EDT_9_2_HL := ai.Toy_podshipnika_rab_kol_EDT_9_2.HL;
AI_Toy_podshipnika_rab_kol_EDT_9_2_LL := ai.Toy_podshipnika_rab_kol_EDT_9_2.LL;
AI_Toy_podshipnika_rab_kol_EDT_9_2_status := DWORD_TO_UDINT(ai.Toy_podshipnika_rab_kol_EDT_9_2.status);
AI_Toy_podshipnika_rab_kol_EDT_9_2_value := ai.Toy_podshipnika_rab_kol_EDT_9_2.value;
AI_Toy_podshipnika_rab_kol_EDT_9_2_HW := ai.Toy_podshipnika_rab_kol_EDT_9_2.HW;
AI_Toy_podshipnika_rab_kol_EDT_9_2_HA := ai.Toy_podshipnika_rab_kol_EDT_9_2.HA;

AI_Toy_podshipnika_nerab_kol_EDT_10_1_HL := ai.Toy_podshipnika_nerab_kol_EDT_10_1.HL;
AI_Toy_podshipnika_nerab_kol_EDT_10_1_LL := ai.Toy_podshipnika_nerab_kol_EDT_10_1.LL;
AI_Toy_podshipnika_nerab_kol_EDT_10_1_status := DWORD_TO_UDINT(ai.Toy_podshipnika_nerab_kol_EDT_10_1.status);
AI_Toy_podshipnika_nerab_kol_EDT_10_1_value := ai.Toy_podshipnika_nerab_kol_EDT_10_1.value;
AI_Toy_podshipnika_nerab_kol_EDT_10_1_HW := ai.Toy_podshipnika_nerab_kol_EDT_10_1.HW;
AI_Toy_podshipnika_nerab_kol_EDT_10_1_HA := ai.Toy_podshipnika_nerab_kol_EDT_10_1.HA;

AI_Toy_podshipnika_nerab_kol_EDT_10_2_HL := ai.Toy_podshipnika_nerab_kol_EDT_10_2.HL;
AI_Toy_podshipnika_nerab_kol_EDT_10_2_LL := ai.Toy_podshipnika_nerab_kol_EDT_10_2.LL;
AI_Toy_podshipnika_nerab_kol_EDT_10_2_status := DWORD_TO_UDINT(ai.Toy_podshipnika_nerab_kol_EDT_10_2.status);
AI_Toy_podshipnika_nerab_kol_EDT_10_2_value := ai.Toy_podshipnika_nerab_kol_EDT_10_2.value;
AI_Toy_podshipnika_nerab_kol_EDT_10_2_HW := ai.Toy_podshipnika_nerab_kol_EDT_10_2.HW;
AI_Toy_podshipnika_nerab_kol_EDT_10_2_HA := ai.Toy_podshipnika_nerab_kol_EDT_10_2.HA;

AI_Tholodnogo_vozduha_ED_kanal_1_HL := ai.Tholodnogo_vozduha_ED_kanal_1.HL;
AI_Tholodnogo_vozduha_ED_kanal_1_LL := ai.Tholodnogo_vozduha_ED_kanal_1.LL;
AI_Tholodnogo_vozduha_ED_kanal_1_status := DWORD_TO_UDINT(ai.Tholodnogo_vozduha_ED_kanal_1.status);
AI_Tholodnogo_vozduha_ED_kanal_1_value := ai.Tholodnogo_vozduha_ED_kanal_1.value;
AI_Tholodnogo_vozduha_ED_kanal_1_HW := ai.Tholodnogo_vozduha_ED_kanal_1.HW;

AI_Tholodnogo_vozduha_ED_kanal_2_HL := ai.Tholodnogo_vozduha_ED_kanal_2.HL;
AI_Tholodnogo_vozduha_ED_kanal_2_LL := ai.Tholodnogo_vozduha_ED_kanal_2.LL;
AI_Tholodnogo_vozduha_ED_kanal_2_status := DWORD_TO_UDINT(ai.Tholodnogo_vozduha_ED_kanal_2.status);
AI_Tholodnogo_vozduha_ED_kanal_2_value := ai.Tholodnogo_vozduha_ED_kanal_2.value;
AI_Tholodnogo_vozduha_ED_kanal_2_HW := ai.Tholodnogo_vozduha_ED_kanal_2.HW;

AI_Tgorjachego_vozduha_ED_kanal_1_HL := ai.Tgorjachego_vozduha_ED_kanal_1.HL;
AI_Tgorjachego_vozduha_ED_kanal_1_LL := ai.Tgorjachego_vozduha_ED_kanal_1.LL;
AI_Tgorjachego_vozduha_ED_kanal_1_status := DWORD_TO_UDINT(ai.Tgorjachego_vozduha_ED_kanal_1.status);
AI_Tgorjachego_vozduha_ED_kanal_1_value := ai.Tgorjachego_vozduha_ED_kanal_1.value;
AI_Tgorjachego_vozduha_ED_kanal_1_HW := ai.Tgorjachego_vozduha_ED_kanal_1.HW;

AI_Tgorjachego_vozduha_ED_kanal_2_HL := ai.Tgorjachego_vozduha_ED_kanal_2.HL;
AI_Tgorjachego_vozduha_ED_kanal_2_LL := ai.Tgorjachego_vozduha_ED_kanal_2.LL;
AI_Tgorjachego_vozduha_ED_kanal_2_status := DWORD_TO_UDINT(ai.Tgorjachego_vozduha_ED_kanal_2.status);
AI_Tgorjachego_vozduha_ED_kanal_2_value := ai.Tgorjachego_vozduha_ED_kanal_2.value;
AI_Tgorjachego_vozduha_ED_kanal_2_HW := ai.Tgorjachego_vozduha_ED_kanal_2.HW;

AI_Tnarujnogo_vozduha_HL := ai.Tnarujnogo_vozduha.HL;
AI_Tnarujnogo_vozduha_LL := ai.Tnarujnogo_vozduha.LL;
AI_Tnarujnogo_vozduha_status := DWORD_TO_UDINT(ai.Tnarujnogo_vozduha.status);
AI_Tnarujnogo_vozduha_value := ai.Tnarujnogo_vozduha.value;
AI_Tnarujnogo_vozduha_HW := ai.Tnarujnogo_vozduha.HW;

AI_Tgaza_na_vhode_H_HL := ai.Tgaza_na_vhode_H.HL;
AI_Tgaza_na_vhode_H_LL := ai.Tgaza_na_vhode_H.LL;
AI_Tgaza_na_vhode_H_status := DWORD_TO_UDINT(ai.Tgaza_na_vhode_H.status);
AI_Tgaza_na_vhode_H_value := ai.Tgaza_na_vhode_H.value;
AI_Tgaza_na_vhode_H_HW := ai.Tgaza_na_vhode_H.HW;

AI_Tgaza_na_vyhode_H_HL := ai.Tgaza_na_vyhode_H.HL;
AI_Tgaza_na_vyhode_H_LL := ai.Tgaza_na_vyhode_H.LL;
AI_Tgaza_na_vyhode_H_status := DWORD_TO_UDINT(ai.Tgaza_na_vyhode_H.status);
AI_Tgaza_na_vyhode_H_value := ai.Tgaza_na_vyhode_H.value;
AI_Tgaza_na_vyhode_H_HW := ai.Tgaza_na_vyhode_H.HW;
AI_Tgaza_na_vyhode_H_HA := ai.Tgaza_na_vyhode_H.HA;

AI_Tmasla_do_AVOM_HL := ai.Tmasla_do_AVOM.HL;
AI_Tmasla_do_AVOM_LL := ai.Tmasla_do_AVOM.LL;
AI_Tmasla_do_AVOM_status := DWORD_TO_UDINT(ai.Tmasla_do_AVOM.status);
AI_Tmasla_do_AVOM_value := ai.Tmasla_do_AVOM.value;
AI_Tmasla_do_AVOM_HW := ai.Tmasla_do_AVOM.HW;

AI_Tmasla_posle_AVOM_HL := ai.Tmasla_posle_AVOM.HL;
AI_Tmasla_posle_AVOM_LL := ai.Tmasla_posle_AVOM.LL;
AI_Tmasla_posle_AVOM_status := DWORD_TO_UDINT(ai.Tmasla_posle_AVOM.status);
AI_Tmasla_posle_AVOM_value := ai.Tmasla_posle_AVOM.value;
AI_Tmasla_posle_AVOM_HW := ai.Tmasla_posle_AVOM.HW;

AI_Tmasla_MB_HL := ai.Tmasla_MB.HL;
AI_Tmasla_MB_LL := ai.Tmasla_MB.LL;
AI_Tmasla_MB_status := DWORD_TO_UDINT(ai.Tmasla_MB.status);
AI_Tmasla_MB_value := ai.Tmasla_MB.value;
AI_Tmasla_MB_HW := ai.Tmasla_MB.HW;

AI_Tmasla_MB_TEN_HL := ai.Tmasla_MB_TEN.HL;
AI_Tmasla_MB_TEN_LL := ai.Tmasla_MB_TEN.LL;
AI_Tmasla_MB_TEN_status := DWORD_TO_UDINT(ai.Tmasla_MB_TEN.status);
AI_Tmasla_MB_TEN_value := ai.Tmasla_MB_TEN.value;
AI_Tmasla_MB_TEN_HW := ai.Tmasla_MB_TEN.HW;

AI_Tshu_HL := ai.Tshu.HL;
AI_Tshu_LL := ai.Tshu.LL;
AI_Tshu_status := DWORD_TO_UDINT(ai.Tshu.status);
AI_Tshu_value := ai.Tshu.value;

AI_Pmaslo_sm_nizkoe_HL := ai.Pmaslo_sm_nizkoe.HL;
AI_Pmaslo_sm_nizkoe_LL := ai.Pmaslo_sm_nizkoe.LL;
AI_Pmaslo_sm_nizkoe_status := DWORD_TO_UDINT(ai.Pmaslo_sm_nizkoe.status);
AI_Pmaslo_sm_nizkoe_value := ai.Pmaslo_sm_nizkoe.value;
AI_Pmaslo_sm_nizkoe_LW := ai.Pmaslo_sm_nizkoe.LW;
AI_Pmaslo_sm_nizkoe_LA := ai.Pmaslo_sm_nizkoe.LA;

AI_Pmaslo_sm_vysokoe_HL := ai.Pmaslo_sm_vysokoe.HL;
AI_Pmaslo_sm_vysokoe_LL := ai.Pmaslo_sm_vysokoe.LL;
AI_Pmaslo_sm_vysokoe_status := DWORD_TO_UDINT(ai.Pmaslo_sm_vysokoe.status);
AI_Pmaslo_sm_vysokoe_value := ai.Pmaslo_sm_vysokoe.value;
AI_Pmaslo_sm_vysokoe_LW := ai.Pmaslo_sm_vysokoe.LW;
AI_Pmaslo_sm_vysokoe_LA := ai.Pmaslo_sm_vysokoe.LA;

AI_Pmasla_posle_GNS_HL := ai.Pmasla_posle_GNS.HL;
AI_Pmasla_posle_GNS_LL := ai.Pmasla_posle_GNS.LL;
AI_Pmasla_posle_GNS_status := DWORD_TO_UDINT(ai.Pmasla_posle_GNS.status);
AI_Pmasla_posle_GNS_value := ai.Pmasla_posle_GNS.value;
AI_Pmasla_posle_GNS_HW := ai.Pmasla_posle_GNS.HW;
AI_Pmasla_posle_GNS_LW := ai.Pmasla_posle_GNS.LW;

AI_Pmasla_posle_NU_HL := ai.Pmasla_posle_NU.HL;
AI_Pmasla_posle_NU_LL := ai.Pmasla_posle_NU.LL;
AI_Pmasla_posle_NU_status := DWORD_TO_UDINT(ai.Pmasla_posle_NU.status);
AI_Pmasla_posle_NU_value := ai.Pmasla_posle_NU.value;
AI_Pmasla_posle_NU_LW := ai.Pmasla_posle_NU.LW;

AI_Pgaza_na_vhode_nagnetatelia_HL := ai.Pgaza_na_vhode_nagnetatelia.HL;
AI_Pgaza_na_vhode_nagnetatelia_LL := ai.Pgaza_na_vhode_nagnetatelia.LL;
AI_Pgaza_na_vhode_nagnetatelia_status := DWORD_TO_UDINT(ai.Pgaza_na_vhode_nagnetatelia.status);
AI_Pgaza_na_vhode_nagnetatelia_value := ai.Pgaza_na_vhode_nagnetatelia.value;
AI_Pgaza_na_vhode_nagnetatelia_LW := ai.Pgaza_na_vhode_nagnetatelia.LW;

AI_Pgaza_na_vyhode_nagnetatelia_HL := ai.Pgaza_na_vyhode_nagnetatelia.HL;
AI_Pgaza_na_vyhode_nagnetatelia_LL := ai.Pgaza_na_vyhode_nagnetatelia.LL;
AI_Pgaza_na_vyhode_nagnetatelia_status := DWORD_TO_UDINT(ai.Pgaza_na_vyhode_nagnetatelia.status);
AI_Pgaza_na_vyhode_nagnetatelia_value := ai.Pgaza_na_vyhode_nagnetatelia.value;
AI_Pgaza_na_vyhode_nagnetatelia_LW := ai.Pgaza_na_vyhode_nagnetatelia.LW;
AI_Pgaza_na_vyhode_nagnetatelia_HA := ai.Pgaza_na_vyhode_nagnetatelia.HA;

AI_Pimpuls_gaz_HL := ai.Pimpuls_gaz.HL;
AI_Pimpuls_gaz_LL := ai.Pimpuls_gaz.LL;
AI_Pimpuls_gaz_status := DWORD_TO_UDINT(ai.Pimpuls_gaz.status);
AI_Pimpuls_gaz_value := ai.Pimpuls_gaz.value;
AI_Pimpuls_gaz_LW := ai.Pimpuls_gaz.LW;

AI_dPgaza_na_maslo_filtre_HL := ai.dPgaza_na_maslo_filtre.HL;
AI_dPgaza_na_maslo_filtre_LL := ai.dPgaza_na_maslo_filtre.LL;
AI_dPgaza_na_maslo_filtre_status := DWORD_TO_UDINT(ai.dPgaza_na_maslo_filtre.status);
AI_dPgaza_na_maslo_filtre_value := ai.dPgaza_na_maslo_filtre.value;
AI_dPgaza_na_maslo_filtre_HW := ai.dPgaza_na_maslo_filtre.HW;

AI_dPgaza_na_konfuzore_HL := ai.dPgaza_na_konfuzore.HL;
AI_dPgaza_na_konfuzore_LL := ai.dPgaza_na_konfuzore.LL;
AI_dPgaza_na_konfuzore_status := DWORD_TO_UDINT(ai.dPgaza_na_konfuzore.status);
AI_dPgaza_na_konfuzore_value := ai.dPgaza_na_konfuzore.value;
AI_dPgaza_na_konfuzore_LW := ai.dPgaza_na_konfuzore.LW;

AI_dPmaslo_gaz_HL := ai.dPmaslo_gaz.HL;
AI_dPmaslo_gaz_LL := ai.dPmaslo_gaz.LL;
AI_dPmaslo_gaz_status := DWORD_TO_UDINT(ai.dPmaslo_gaz.status);
AI_dPmaslo_gaz_value := ai.dPmaslo_gaz.value;
AI_dPmaslo_gaz_LW := ai.dPmaslo_gaz.LW;
AI_dPmaslo_gaz_LA := ai.dPmaslo_gaz.LA;

AI_Os_sdvig_nagnetatelja_plus_HL := ai.Os_sdvig_nagnetatelja_plus.HL;
AI_Os_sdvig_nagnetatelja_plus_LL := ai.Os_sdvig_nagnetatelja_plus.LL;
AI_Os_sdvig_nagnetatelja_plus_status := DWORD_TO_UDINT(ai.Os_sdvig_nagnetatelja_plus.status);
AI_Os_sdvig_nagnetatelja_plus_value := ai.Os_sdvig_nagnetatelja_plus.value;
AI_Os_sdvig_nagnetatelja_plus_HW := ai.Os_sdvig_nagnetatelja_plus.HW;
AI_Os_sdvig_nagnetatelja_plus_HA := ai.Os_sdvig_nagnetatelja_plus.HA;

AI_Os_sdvig_nagnetatelja_minus_HL := ai.Os_sdvig_nagnetatelja_minus.HL;
AI_Os_sdvig_nagnetatelja_minus_LL := ai.Os_sdvig_nagnetatelja_minus.LL;
AI_Os_sdvig_nagnetatelja_minus_status := DWORD_TO_UDINT(ai.Os_sdvig_nagnetatelja_minus.status);
AI_Os_sdvig_nagnetatelja_minus_value := ai.Os_sdvig_nagnetatelja_minus.value;
AI_Os_sdvig_nagnetatelja_minus_LW := ai.Os_sdvig_nagnetatelja_minus.LW;
AI_Os_sdvig_nagnetatelja_minus_LA := ai.Os_sdvig_nagnetatelja_minus.LA;

AI_Yroven_masla_MB_HL := ai.Yroven_masla_MB.HL;
AI_Yroven_masla_MB_LL := ai.Yroven_masla_MB.LL;
AI_Yroven_masla_MB_status := DWORD_TO_UDINT(ai.Yroven_masla_MB.status);
AI_Yroven_masla_MB_value := ai.Yroven_masla_MB.value;
AI_Yroven_masla_MB_LW := ai.Yroven_masla_MB.LW;

AI_Kontrol_per_220V_HL := ai.Kontrol_per_220V.HL;
AI_Kontrol_per_220V_LL := ai.Kontrol_per_220V.LL;
AI_Kontrol_per_220V_status := DWORD_TO_UDINT(ai.Kontrol_per_220V.status);
AI_Kontrol_per_220V_value := ai.Kontrol_per_220V.value;
AI_Kontrol_per_220V_HW := ai.Kontrol_per_220V.HW;
AI_Kontrol_per_220V_LW := ai.Kontrol_per_220V.LW;

AI_Kontrol_post_220V_HL := ai.Kontrol_post_220V.HL;
AI_Kontrol_post_220V_LL := ai.Kontrol_post_220V.LL;
AI_Kontrol_post_220V_status := DWORD_TO_UDINT(ai.Kontrol_post_220V.status);
AI_Kontrol_post_220V_value := ai.Kontrol_post_220V.value;
AI_Kontrol_post_220V_HW := ai.Kontrol_post_220V.HW;
AI_Kontrol_post_220V_LW := ai.Kontrol_post_220V.LW;

AI_Tok_statora_HL := ai.Tok_statora.HL;
AI_Tok_statora_LL := ai.Tok_statora.LL;
AI_Tok_statora_status := DWORD_TO_UDINT(ai.Tok_statora.status);
AI_Tok_statora_value := ai.Tok_statora.value;
AI_Tok_statora_LW := ai.Tok_statora.LW;

AI_Vibro_skorost_OPED_T1_HL := ai.Vibro_skorost_OPED_T1.HL;
AI_Vibro_skorost_OPED_T1_LL := ai.Vibro_skorost_OPED_T1.LL;
AI_Vibro_skorost_OPED_T1_status := DWORD_TO_UDINT(ai.Vibro_skorost_OPED_T1.status);
AI_Vibro_skorost_OPED_T1_value := ai.Vibro_skorost_OPED_T1.value;
AI_Vibro_skorost_OPED_T1_HW := ai.Vibro_skorost_OPED_T1.HW;
AI_Vibro_skorost_OPED_T1_HA := ai.Vibro_skorost_OPED_T1.HA;

AI_Vibro_skorost_OYPED_T2_HL := ai.Vibro_skorost_OYPED_T2.HL;
AI_Vibro_skorost_OYPED_T2_LL := ai.Vibro_skorost_OYPED_T2.LL;
AI_Vibro_skorost_OYPED_T2_status := DWORD_TO_UDINT(ai.Vibro_skorost_OYPED_T2.status);
AI_Vibro_skorost_OYPED_T2_value := ai.Vibro_skorost_OYPED_T2.value;
AI_Vibro_skorost_OYPED_T2_HW := ai.Vibro_skorost_OYPED_T2.HW;
AI_Vibro_skorost_OYPED_T2_HA := ai.Vibro_skorost_OYPED_T2.HA;

AI_Vibro_skorost_OYP_kolesa_ED_T3_HL := ai.Vibro_skorost_OYP_kolesa_ED_T3.HL;
AI_Vibro_skorost_OYP_kolesa_ED_T3_LL := ai.Vibro_skorost_OYP_kolesa_ED_T3.LL;
AI_Vibro_skorost_OYP_kolesa_ED_T3_status := DWORD_TO_UDINT(ai.Vibro_skorost_OYP_kolesa_ED_T3.status);
AI_Vibro_skorost_OYP_kolesa_ED_T3_value := ai.Vibro_skorost_OYP_kolesa_ED_T3.value;
AI_Vibro_skorost_OYP_kolesa_ED_T3_HW := ai.Vibro_skorost_OYP_kolesa_ED_T3.HW;
AI_Vibro_skorost_OYP_kolesa_ED_T3_HA := ai.Vibro_skorost_OYP_kolesa_ED_T3.HA;

AI_Vibro_skorost_OP_kolesa_RH_T4_HL := ai.Vibro_skorost_OP_kolesa_RH_T4.HL;
AI_Vibro_skorost_OP_kolesa_RH_T4_LL := ai.Vibro_skorost_OP_kolesa_RH_T4.LL;
AI_Vibro_skorost_OP_kolesa_RH_T4_status := DWORD_TO_UDINT(ai.Vibro_skorost_OP_kolesa_RH_T4.status);
AI_Vibro_skorost_OP_kolesa_RH_T4_value := ai.Vibro_skorost_OP_kolesa_RH_T4.value;
AI_Vibro_skorost_OP_kolesa_RH_T4_HW := ai.Vibro_skorost_OP_kolesa_RH_T4.HW;
AI_Vibro_skorost_OP_kolesa_RH_T4_HA := ai.Vibro_skorost_OP_kolesa_RH_T4.HA;

AI_Vibro_skorost_OP_shesterni_RED_T5_HL := ai.Vibro_skorost_OP_shesterni_RED_T5.HL;
AI_Vibro_skorost_OP_shesterni_RED_T5_LL := ai.Vibro_skorost_OP_shesterni_RED_T5.LL;
AI_Vibro_skorost_OP_shesterni_RED_T5_status := DWORD_TO_UDINT(ai.Vibro_skorost_OP_shesterni_RED_T5.status);
AI_Vibro_skorost_OP_shesterni_RED_T5_value := ai.Vibro_skorost_OP_shesterni_RED_T5.value;
AI_Vibro_skorost_OP_shesterni_RED_T5_HW := ai.Vibro_skorost_OP_shesterni_RED_T5.HW;
AI_Vibro_skorost_OP_shesterni_RED_T5_HA := ai.Vibro_skorost_OP_shesterni_RED_T5.HA;

AI_Vibro_skorost_OP_shesterni_RED_T6_HL := ai.Vibro_skorost_OP_shesterni_RED_T6.HL;
AI_Vibro_skorost_OP_shesterni_RED_T6_LL := ai.Vibro_skorost_OP_shesterni_RED_T6.LL;
AI_Vibro_skorost_OP_shesterni_RED_T6_status := DWORD_TO_UDINT(ai.Vibro_skorost_OP_shesterni_RED_T6.status);
AI_Vibro_skorost_OP_shesterni_RED_T6_value := ai.Vibro_skorost_OP_shesterni_RED_T6.value;
AI_Vibro_skorost_OP_shesterni_RED_T6_HW := ai.Vibro_skorost_OP_shesterni_RED_T6.HW;
AI_Vibro_skorost_OP_shesterni_RED_T6_HA := ai.Vibro_skorost_OP_shesterni_RED_T6.HA;

(* ---- OPC_algoritms_get.st ---- *)
FUNCTION_BLOCK OPC_algoritms_get

VAR_EXTERNAL
	algoritms_autoNu : UINT;
	algoritms_AutoPns : UINT;
	algoritms_AutoAvom : UINT;
	algoritms_AutoTen : UINT;
	algoritms_AntiPompag : UINT;
	algoritms_testIm : UINT;
	algoritms_TestProtection : UINT;
	algoritms_Remont : UINT;
	algoritms_ppu : UINT;
	algoritms_puskOilSystem : UINT;
	algoritms_engineRun : UINT;
	algoritms_filling : UINT;
	algoritms_LineToRing : UINT;
	algoritms_RingToLine : UINT;
	algoritms_Apusk : UINT;
	algoritms_SemiAutoPusk : UINT;
	algoritms_no : UINT;
	algoritms_vibegPNS : UINT;
	algoritms_ao : UINT;
	algoritms_testPms : UINT;
	algoritms_testdPmg : UINT;
	algoritms_puskV : UINT;
	algoritms_puskK : UINT;
	algoritms_Pusk_F_faza1 : UINT;
	algoritms_Pusk_F_faza2 : UINT;
	algoritms_Pusk_TH_faza : UINT;
	algoritms_Prov_PMS_ALG : UINT;
	algoritms_Prov_opressovka_ALG : UINT;
	algoritms_Pusk_SEC_faza_chastotny : UINT;
	algoritms_Pusk_SEC_faza_reactor : UINT;
	algoritms : AlgoritmsConfig;
END_VAR

algoritms.autoNu.inCommand_ARM := UINT_TO_WORD(algoritms_autoNu);

algoritms.AutoPns.inCommand_ARM := UINT_TO_WORD(algoritms_AutoPns);

algoritms.AutoAvom.inCommand_ARM := UINT_TO_WORD(algoritms_AutoAvom);

algoritms.AutoTen.inCommand_ARM := UINT_TO_WORD(algoritms_AutoTen);

algoritms.AntiPompag.inCommand_ARM := UINT_TO_WORD(algoritms_AntiPompag);

algoritms.testIm.inCommand_ARM := UINT_TO_WORD(algoritms_testIm);

algoritms.TestProtection.inCommand_ARM := UINT_TO_WORD(algoritms_TestProtection);

algoritms.Remont.inCommand_ARM := UINT_TO_WORD(algoritms_Remont);

algoritms.ppu.inCommand_ARM := UINT_TO_WORD(algoritms_ppu);

algoritms.puskOilSystem.inCommand_ARM := UINT_TO_WORD(algoritms_puskOilSystem);

algoritms.engineRun.inCommand_ARM := UINT_TO_WORD(algoritms_engineRun);

algoritms.filling.inCommand_ARM := UINT_TO_WORD(algoritms_filling);

algoritms.LineToRing.inCommand_ARM := UINT_TO_WORD(algoritms_LineToRing);

algoritms.RingToLine.inCommand_ARM := UINT_TO_WORD(algoritms_RingToLine);

algoritms.Apusk.inCommand_ARM := UINT_TO_WORD(algoritms_Apusk);

algoritms.SemiAutoPusk.inCommand_ARM := UINT_TO_WORD(algoritms_SemiAutoPusk);

algoritms.no.inCommand_ARM := UINT_TO_WORD(algoritms_no);

algoritms.vibegPNS.inCommand_ARM := UINT_TO_WORD(algoritms_vibegPNS);

algoritms.ao.inCommand_ARM := UINT_TO_WORD(algoritms_ao);

algoritms.testPms.inCommand_ARM := UINT_TO_WORD(algoritms_testPms);

algoritms.testdPmg.inCommand_ARM := UINT_TO_WORD(algoritms_testdPmg);

algoritms.puskV.inCommand_ARM := UINT_TO_WORD(algoritms_puskV);

algoritms.puskK.inCommand_ARM := UINT_TO_WORD(algoritms_puskK);

algoritms.Pusk_F_faza1.inCommand_ARM := UINT_TO_WORD(algoritms_Pusk_F_faza1);

algoritms.Pusk_F_faza2.inCommand_ARM := UINT_TO_WORD(algoritms_Pusk_F_faza2);

algoritms.Pusk_TH_faza.inCommand_ARM := UINT_TO_WORD(algoritms_Pusk_TH_faza);

algoritms.Prov_PMS_ALG.inCommand_ARM := UINT_TO_WORD(algoritms_Prov_PMS_ALG);

algoritms.Prov_opressovka_ALG.inCommand_ARM := UINT_TO_WORD(algoritms_Prov_opressovka_ALG);

algoritms.Pusk_SEC_faza_chastotny.inCommand_ARM := UINT_TO_WORD(algoritms_Pusk_SEC_faza_chastotny);

algoritms.Pusk_SEC_faza_reactor.inCommand_ARM := UINT_TO_WORD(algoritms_Pusk_SEC_faza_reactor);

(* ---- OPC_algoritms_set.st ---- *)
FUNCTION_BLOCK OPC_algoritms_set

VAR_EXTERNAL
	algoritms : AlgoritmsConfig;
	algManager_Mode : UINT;
	algoritms_AutoAvom_status : UDINT;
	algoritms_AutoPns_OffTimer : UINT;
	algoritms_AutoPns_OnTimer : UINT;
	algoritms_AutoPns_status : UDINT;
	algoritms_AutoTen_status : UDINT;
	algoritms_Remont_status : UDINT;
	algoritms_TestProtection_status : UDINT;
	algoritms_autoNu_NotHasRezervNU : BOOL;
	algoritms_autoNu_status : UDINT;
	algoritms_Pusk_SEC_faza_reactor_Top : UDINT;
	algoritms_Pusk_SEC_faza_reactor_Error : UDINT;
	algoritms_Pusk_SEC_faza_reactor_Start : UDINT;
	algoritms_Pusk_SEC_faza_reactor_status : UDINT;
	algoritms_Pusk_SEC_faza_chastotny_Top : UDINT;
	algoritms_Pusk_SEC_faza_chastotny_Error : UDINT;
	algoritms_Pusk_SEC_faza_chastotny_Start : UDINT;
	algoritms_Pusk_SEC_faza_chastotny_status : UDINT;
	algoritms_Prov_opressovka_ALG_Top : UDINT;
	algoritms_Prov_opressovka_ALG_Error : UDINT;
	algoritms_Prov_opressovka_ALG_Start : UDINT;
	algoritms_Prov_opressovka_ALG_status : UDINT;
	algoritms_Prov_PMS_ALG_Top : UDINT;
	algoritms_Prov_PMS_ALG_Error : UDINT;
	algoritms_Prov_PMS_ALG_Start : UDINT;
	algoritms_Prov_PMS_ALG_status : UDINT;
	algoritms_Pusk_TH_faza_Top : UDINT;
	algoritms_Pusk_TH_faza_Error : UDINT;
	algoritms_Pusk_TH_faza_Start : UDINT;
	algoritms_Pusk_TH_faza_status : UDINT;
	algoritms_Pusk_F_faza2_Top : UDINT;
	algoritms_Pusk_F_faza2_Error : UDINT;
	algoritms_Pusk_F_faza2_Start : UDINT;
	algoritms_Pusk_F_faza2_status : UDINT;
	algoritms_Pusk_F_faza1_Top : UDINT;
	algoritms_Pusk_F_faza1_Error : UDINT;
	algoritms_Pusk_F_faza1_Start : UDINT;
	algoritms_Pusk_F_faza1_status : UDINT;
	algoritms_puskOilSystem_Error : UDINT;
	algoritms_puskOilSystem_Start : UDINT;
	algoritms_puskOilSystem_Top : UDINT;
	algoritms_puskOilSystem_status : UDINT;
	algoritms_testIm_status : UDINT;
	algoritms_vibegPNS_Error : UDINT;
	algoritms_vibegPNS_Start : UDINT;
	algoritms_vibegPNS_Top : UDINT;
	algoritms_vibegPNS_algContinue_status : UDINT;
	algoritms_vibegPNS_status : UDINT;
	algoritms_vibegPNS_waitVibeg_timer : UINT;
	protectManager_protectionInRemont : BOOL;
	algManager : struct_AlgoritmsManager;
	protectManager : struct_ProtectionsManager;
	NotHasRezervNU : BOOL;
	AlgTimers : struct_AlgTimers;
	AlgQuestions : AlgoritmsQuestions;
	algoritms_Apusk_Error : UDINT;
	algoritms_Apusk_Start : UDINT;
	algoritms_Apusk_Top : UDINT;
	algoritms_Apusk_status : UDINT;
	algoritms_RingToLine_Error : UDINT;
	algoritms_RingToLine_Start : UDINT;
	algoritms_RingToLine_Top : UDINT;
	algoritms_RingToLine_status : UDINT;
	algoritms_ao_Error : UDINT;
	algoritms_ao_Start : UDINT;
	algoritms_ao_Top : UDINT;
	algoritms_ao_status : UDINT;
	algoritms_ao_waitKran_timer : UINT;
	algoritms_engineRun_BreakPuskTimer_timer : UINT;
	algoritms_engineRun_Error : UDINT;
	algoritms_engineRun_Start : UDINT;
	algoritms_engineRun_Top : UDINT;
	algoritms_engineRun_status : UDINT;
	algoritms_filling_BreakPuskTimer_timer : UINT;
	algoritms_filling_Error : UDINT;
	algoritms_filling_Start : UDINT;
	algoritms_filling_Top : UDINT;
	algoritms_filling_status : UDINT;
	algoritms_filling_waitAfterKran4_timer : UINT;
	algoritms_filling_waitAfterKran5_timer : UINT;
	algoritms_no_Error : UDINT;
	algoritms_no_Start : UDINT;
	algoritms_no_Top : UDINT;
	algoritms_no_status : UDINT;
	algoritms_no_waitCloseKran_timer : UINT;
	algoritms_ppu_Error : UDINT;
	algoritms_ppu_Start : UDINT;
	algoritms_ppu_Top : UDINT;
	algoritms_ppu_status : UDINT;
	algoritms_puskK_Error : UDINT;
	algoritms_puskK_Start : UDINT;
	algoritms_puskK_Top : UDINT;
	algoritms_puskK_questionFilling_status : UDINT;
	algoritms_puskK_questionUnload_status : UDINT;
	algoritms_puskK_status : UDINT;
	algoritms_autoNu_Start : UDINT;
	algoritms_autoNu_Error : UDINT;
	algoritms_autoNu_Top : UDINT;
	algoritms_AutoAvom_Start : UDINT;
	algoritms_AutoAvom_Error : UDINT;
	algoritms_AutoAvom_Top : UDINT;
	algoritms_puskK_wait720_timer : UINT;
	algoritms_puskOilSystem_BreakPuskTimer_Poil_timer : UINT;
	algoritms_puskOilSystem_BreakPuskTimer_dPmg_timer : UINT;
	algoritms_testPms_BreakTest_timer : UINT;
	algoritms_testPms_Error : UDINT;
	algoritms_testPms_Start : UDINT;
	algoritms_testPms_Top : UDINT;
	algoritms_testPms_algContinue_status : UDINT;
	algoritms_testPms_status : UDINT;
	algoritms_testdPmg_BreakTest_timer : UINT;
	algoritms_testdPmg_Error : UDINT;
	algoritms_testdPmg_Start : UDINT;
	algoritms_testdPmg_Top : UDINT;
	algoritms_testdPmg_algContinue_status : UDINT;
	algoritms_testdPmg_status : UDINT;
END_VAR

(* OPC Set - algoritms. Запись текущих состояний тэгов _______________________________________________________*)

algManager_Mode := algManager.mode;

protectManager_protectionInRemont:= protectManager.protectionInRemont;

algoritms_autoNu_NotHasRezervNU:= NotHasRezervNU;

algoritms_no_Start	:= DWORD_TO_UDINT(algoritms.no.Start);
algoritms_no_Error	:= DWORD_TO_UDINT(algoritms.no.Error);
algoritms_no_Top	:= DWORD_TO_UDINT(algoritms.no.Top);
algoritms_no_status	:= DWORD_TO_UDINT(algoritms.no.status);
algoritms_no_waitCloseKran_timer	:= AlgTimers.NO_waitCloseKran;

algoritms_ao_Start	:= DWORD_TO_UDINT(algoritms.ao.Start);
algoritms_ao_Error	:= DWORD_TO_UDINT(algoritms.ao.Error);
algoritms_ao_Top	:= DWORD_TO_UDINT(algoritms.ao.Top);
algoritms_ao_status	:= DWORD_TO_UDINT(algoritms.ao.status);
algoritms_ao_waitKran_timer	:= AlgTimers.AO_waitKran;

algoritms_vibegPNS_Start		:= DWORD_TO_UDINT(algoritms.vibegPNS.Start);
algoritms_vibegPNS_Error		:= DWORD_TO_UDINT(algoritms.vibegPNS.Error);
algoritms_vibegPNS_Top		:= DWORD_TO_UDINT(algoritms.vibegPNS.Top);
algoritms_vibegPNS_status		:= DWORD_TO_UDINT(algoritms.vibegPNS.status);
algoritms_vibegPNS_waitVibeg_timer	:= AlgTimers.vibegPNS_Timer;
algoritms_vibegPNS_algContinue_status	:= DWORD_TO_UDINT(AlgQuestions.vibegPNS_algContinue.status);

algoritms_testPms_Start		:= DWORD_TO_UDINT(algoritms.testPms.Start);
algoritms_testPms_Error		:= DWORD_TO_UDINT(algoritms.testPms.Error);
algoritms_testPms_Top		:= DWORD_TO_UDINT(algoritms.testPms.Top);
algoritms_testPms_status		:= DWORD_TO_UDINT(algoritms.testPms.status);
algoritms_testPms_algContinue_status	:= DWORD_TO_UDINT(AlgQuestions.testPms_algContinue.status);
algoritms_testPms_BreakTest_timer	:= AlgTimers.testPms_BreakTest;

algoritms_testdPmg_Start		:= DWORD_TO_UDINT(algoritms.testdPmg.Start);
algoritms_testdPmg_Error		:= DWORD_TO_UDINT(algoritms.testdPmg.Error);
algoritms_testdPmg_Top		:= DWORD_TO_UDINT(algoritms.testdPmg.Top);
algoritms_testdPmg_status		:= DWORD_TO_UDINT(algoritms.testdPmg.status);
algoritms_testdPmg_algContinue_status	:= DWORD_TO_UDINT(AlgQuestions.testdPmg_algContinue.status);
algoritms_testdPmg_BreakTest_timer	:= AlgTimers.testdPmg_BreakTest;

algoritms_testIm_status	:= DWORD_TO_UDINT(algoritms.testIm.status);

algoritms_ppu_status	:= DWORD_TO_UDINT(algoritms.ppu.status);
algoritms_ppu_Start	          := DWORD_TO_UDINT(algoritms.ppu.Start);
algoritms_ppu_Error	          := DWORD_TO_UDINT(algoritms.ppu.Error);
algoritms_ppu_Top	          := DWORD_TO_UDINT(algoritms.ppu.Top);

algoritms_puskOilSystem_status			:= DWORD_TO_UDINT(algoritms.puskOilSystem.status);
algoritms_puskOilSystem_Start				:= DWORD_TO_UDINT(algoritms.puskOilSystem.Start);
algoritms_puskOilSystem_Error				:= DWORD_TO_UDINT(algoritms.puskOilSystem.Error);
algoritms_puskOilSystem_Top				:= DWORD_TO_UDINT(algoritms.puskOilSystem.Top);
algoritms_puskOilSystem_BreakPuskTimer_Poil_timer	          := AlgTimers.puskOilSystem_BreakPuskTimer_Poil;

algoritms_engineRun_status			:= DWORD_TO_UDINT(algoritms.engineRun.status);
algoritms_engineRun_Start			:= DWORD_TO_UDINT(algoritms.engineRun.Start);
algoritms_engineRun_Error			:= DWORD_TO_UDINT(algoritms.engineRun.Error);
algoritms_engineRun_Top			:= DWORD_TO_UDINT(algoritms.engineRun.Top);
algoritms_engineRun_BreakPuskTimer_timer	:= AlgTimers.engineRun_BreakPuskTimer;

algoritms_filling_status		:= DWORD_TO_UDINT(algoritms.filling.status);
algoritms_filling_Start		:= DWORD_TO_UDINT(algoritms.filling.Start);
algoritms_filling_Error		:= DWORD_TO_UDINT(algoritms.filling.Error);
algoritms_filling_Top		:= DWORD_TO_UDINT(algoritms.filling.Top);
algoritms_filling_BreakPuskTimer_timer	:= AlgTimers.filling_BreakPuskTimer;
algoritms_filling_waitAfterKran4_timer	:= AlgTimers.filling_waitAfterKran4;
algoritms_filling_waitAfterKran5_timer	:= AlgTimers.filling_waitAfterKran5;

algoritms_RingToLine_status	:= DWORD_TO_UDINT(algoritms.RingToLine.status);
algoritms_RingToLine_Start	:= DWORD_TO_UDINT(algoritms.RingToLine.Start);
algoritms_RingToLine_Error	:= DWORD_TO_UDINT(algoritms.RingToLine.Error);
algoritms_RingToLine_Top	:= DWORD_TO_UDINT(algoritms.RingToLine.Top);

algoritms_AutoPns_status	:= DWORD_TO_UDINT(algoritms.AutoPns.status);
algoritms_AutoPns_OnTimer	:= AlgTimers.AutoPns_OnTimer;
algoritms_AutoPns_OffTimer	:= AlgTimers.AutoPns_OffTimer;

algoritms_autoNu_status	:= DWORD_TO_UDINT(algoritms.autoNu.status);
algoritms_autoNu_Start	:= DWORD_TO_UDINT(algoritms.autoNu.Start);
algoritms_autoNu_Error	:= DWORD_TO_UDINT(algoritms.autoNu.Error);
algoritms_autoNu_Top	:= DWORD_TO_UDINT(algoritms.autoNu.Top);

algoritms_AutoAvom_status	:= DWORD_TO_UDINT(algoritms.AutoAvom.status);
algoritms_AutoAvom_Start	:= DWORD_TO_UDINT(algoritms.AutoAvom.Start);
algoritms_AutoAvom_Error	:= DWORD_TO_UDINT(algoritms.AutoAvom.Error);
algoritms_AutoAvom_Top	:= DWORD_TO_UDINT(algoritms.AutoAvom.Top);

algoritms_Pusk_F_faza1_status	:= DWORD_TO_UDINT(algoritms.Pusk_F_faza1.status);
algoritms_Pusk_F_faza1_Start	:= DWORD_TO_UDINT(algoritms.Pusk_F_faza1.Start);
algoritms_Pusk_F_faza1_Error	:= DWORD_TO_UDINT(algoritms.Pusk_F_faza1.Error);
algoritms_Pusk_F_faza1_Top	:= DWORD_TO_UDINT(algoritms.Pusk_F_faza1.Top);

algoritms_Pusk_F_faza2_status	:= DWORD_TO_UDINT(algoritms.Pusk_F_faza2.status);
algoritms_Pusk_F_faza2_Start	:= DWORD_TO_UDINT(algoritms.Pusk_F_faza2.Start);
algoritms_Pusk_F_faza2_Error	:= DWORD_TO_UDINT(algoritms.Pusk_F_faza2.Error);
algoritms_Pusk_F_faza2_Top	:= DWORD_TO_UDINT(algoritms.Pusk_F_faza2.Top);

algoritms_Pusk_TH_faza_status	:= DWORD_TO_UDINT(algoritms.Pusk_TH_faza.status);
algoritms_Pusk_TH_faza_Start	:= DWORD_TO_UDINT(algoritms.Pusk_TH_faza.Start);
algoritms_Pusk_TH_faza_Error	:= DWORD_TO_UDINT(algoritms.Pusk_TH_faza.Error);
algoritms_Pusk_TH_faza_Top	:= DWORD_TO_UDINT(algoritms.Pusk_TH_faza.Top);

algoritms_Prov_PMS_ALG_status	:= DWORD_TO_UDINT(algoritms.Prov_PMS_ALG.status);
algoritms_Prov_PMS_ALG_Start	:= DWORD_TO_UDINT(algoritms.Prov_PMS_ALG.Start);
algoritms_Prov_PMS_ALG_Error	:= DWORD_TO_UDINT(algoritms.Prov_PMS_ALG.Error);
algoritms_Prov_PMS_ALG_Top	:= DWORD_TO_UDINT(algoritms.Prov_PMS_ALG.Top);

algoritms_Prov_opressovka_ALG_status	:= DWORD_TO_UDINT(algoritms.Prov_opressovka_ALG.status);
algoritms_Prov_opressovka_ALG_Start	:= DWORD_TO_UDINT(algoritms.Prov_opressovka_ALG.Start);
algoritms_Prov_opressovka_ALG_Error	:= DWORD_TO_UDINT(algoritms.Prov_opressovka_ALG.Error);
algoritms_Prov_opressovka_ALG_Top	:= DWORD_TO_UDINT(algoritms.Prov_opressovka_ALG.Top);

algoritms_Pusk_SEC_faza_chastotny_status	:= DWORD_TO_UDINT(algoritms.Pusk_SEC_faza_chastotny.status);
algoritms_Pusk_SEC_faza_chastotny_Start	:= DWORD_TO_UDINT(algoritms.Pusk_SEC_faza_chastotny.Start);
algoritms_Pusk_SEC_faza_chastotny_Error	:= DWORD_TO_UDINT(algoritms.Pusk_SEC_faza_chastotny.Error);
algoritms_Pusk_SEC_faza_chastotny_Top	:= DWORD_TO_UDINT(algoritms.Pusk_SEC_faza_chastotny.Top);

algoritms_Pusk_SEC_faza_reactor_status	:= DWORD_TO_UDINT(algoritms.Pusk_SEC_faza_reactor.status);
algoritms_Pusk_SEC_faza_reactor_Start	:= DWORD_TO_UDINT(algoritms.Pusk_SEC_faza_reactor.Start);
algoritms_Pusk_SEC_faza_reactor_Error	:= DWORD_TO_UDINT(algoritms.Pusk_SEC_faza_reactor.Error);
algoritms_Pusk_SEC_faza_reactor_Top	:= DWORD_TO_UDINT(algoritms.Pusk_SEC_faza_reactor.Top);

algoritms_Remont_status	:= DWORD_TO_UDINT(algoritms.Remont.status);

algoritms_AutoTen_status	:= DWORD_TO_UDINT(algoritms.AutoTen.status);

(* ---- OPC_IM_GET.st ---- *)
FUNCTION_BLOCK OPC_IM_GET

VAR_EXTERNAL
	IM : ImConfig;
	IM_Kran1_status : UDINT;
	IM_Kran1_inCommand_ARM : UINT;
	IM_Kran2_status : UDINT;
	IM_Kran2_inCommand_ARM : UINT;
	IM_Kran3_status : UDINT;
	IM_Kran3_inCommand_ARM : UINT;
	IM_Kran3b_status : UDINT;
	IM_Kran3b_inCommand_ARM : UINT;
	IM_Kran4_status : UDINT;
	IM_Kran4_inCommand_ARM : UINT;
	IM_Kran5_status : UDINT;
	IM_Kran5_inCommand_ARM : UINT;
	IM_Kran6_status : UDINT;
	IM_Kran6_inCommand_ARM : UINT;
	IM_nu1_status : UDINT;
	IM_nu1_inCommand_ARM : UINT;
	IM_nu2_status : UDINT;
	IM_nu2_inCommand_ARM : UINT;
	IM_pns_status : UDINT;
	IM_pns_inCommand_ARM : UINT;
	IM_v1_Avom_status : UDINT;
	IM_v1_Avom_inCommand_ARM : UINT;
	IM_v2_Avom_status : UDINT;
	IM_v2_Avom_inCommand_ARM : UINT;
	IM_v3_Avom_status : UDINT;
	IM_v3_Avom_inCommand_ARM : UINT;
	IM_v4_Avom_status : UDINT;
	IM_v4_Avom_inCommand_ARM : UINT;
	IM_mv_status : UDINT;
	IM_mv_inCommand_ARM : UINT;
	IM_KaloriferAVOM_status : UDINT;
	IM_KaloriferAVOM_inCommand_ARM : UINT;
	IM_CMN_status : UDINT;
	IM_CMN_inCommand_ARM : UINT;
	IM_TEN_kollectora_status : UDINT;
	IM_TEN_kollectora_inCommand_ARM : UINT;
	IM_TEN_MB_status : UDINT;
	IM_TEN_MB_inCommand_ARM : UINT;
END_VAR

IM.Kran1.inCommand_ARM := UINT_TO_WORD(IM_Kran1_inCommand_ARM);

IM.Kran2.inCommand_ARM := UINT_TO_WORD(IM_Kran2_inCommand_ARM);

IM.Kran3.inCommand_ARM := UINT_TO_WORD(IM_Kran3_inCommand_ARM);

IM.Kran3b.inCommand_ARM := UINT_TO_WORD(IM_Kran3b_inCommand_ARM);

IM.Kran4.inCommand_ARM := UINT_TO_WORD(IM_Kran4_inCommand_ARM);

IM.Kran5.inCommand_ARM := UINT_TO_WORD(IM_Kran5_inCommand_ARM);

IM.Kran6.inCommand_ARM := UINT_TO_WORD(IM_Kran6_inCommand_ARM);

IM.nu1.inCommand_ARM := UINT_TO_WORD(IM_nu1_inCommand_ARM);

IM.nu2.inCommand_ARM := UINT_TO_WORD(IM_nu2_inCommand_ARM);

IM.pns.inCommand_ARM := UINT_TO_WORD(IM_pns_inCommand_ARM);

IM.v1_Avom.inCommand_ARM := UINT_TO_WORD(IM_v1_Avom_inCommand_ARM);

IM.v2_Avom.inCommand_ARM := UINT_TO_WORD(IM_v2_Avom_inCommand_ARM);

IM.v3_Avom.inCommand_ARM := UINT_TO_WORD(IM_v3_Avom_inCommand_ARM);

IM.v4_Avom.inCommand_ARM := UINT_TO_WORD(IM_v4_Avom_inCommand_ARM);

IM.mv.inCommand_ARM := UINT_TO_WORD(IM_mv_inCommand_ARM);

IM.KaloriferAVOM.inCommand_ARM := UINT_TO_WORD(IM_KaloriferAVOM_inCommand_ARM);

IM.CMN.inCommand_ARM := UINT_TO_WORD(IM_CMN_inCommand_ARM);

IM.TEN_kollectora.inCommand_ARM := UINT_TO_WORD(IM_TEN_kollectora_inCommand_ARM);

IM.TEN_MB.inCommand_ARM := UINT_TO_WORD(IM_TEN_MB_inCommand_ARM);

(* ---- OPC_IM_SET.st ---- *)
FUNCTION_BLOCK OPC_IM_SET

VAR_EXTERNAL
	Im : ImConfig;
	IM_Kran1_status : UDINT;
	IM_Kran1_inCommand_ARM : UINT;
	IM_Kran2_status : UDINT;
	IM_Kran2_inCommand_ARM : UINT;
	IM_Kran3_status : UDINT;
	IM_Kran3_inCommand_ARM : UINT;
	IM_Kran3b_status : UDINT;
	IM_Kran3b_inCommand_ARM : UINT;
	IM_Kran4_status : UDINT;
	IM_Kran4_inCommand_ARM : UINT;
	IM_Kran5_status : UDINT;
	IM_Kran5_inCommand_ARM : UINT;
	IM_Kran6_status : UDINT;
	IM_Kran6_inCommand_ARM : UINT;
	IM_nu1_status : UDINT;
	IM_nu1_inCommand_ARM : UINT;
	IM_nu2_status : UDINT;
	IM_nu2_inCommand_ARM : UINT;
	IM_pns_status : UDINT;
	IM_pns_inCommand_ARM : UINT;
	IM_v1_Avom_status : UDINT;
	IM_v1_Avom_inCommand_ARM : UINT;
	IM_v2_Avom_status : UDINT;
	IM_v2_Avom_inCommand_ARM : UINT;
	IM_v3_Avom_status : UDINT;
	IM_v3_Avom_inCommand_ARM : UINT;
	IM_v4_Avom_status : UDINT;
	IM_v4_Avom_inCommand_ARM : UINT;
	IM_mv_status : UDINT;
	IM_mv_inCommand_ARM : UINT;
	IM_KaloriferAVOM_status : UDINT;
	IM_KaloriferAVOM_inCommand_ARM : UINT;
	IM_CMN_status : UDINT;
	IM_CMN_inCommand_ARM : UINT;
	IM_TEN_kollectora_status : UDINT;
	IM_TEN_kollectora_inCommand_ARM : UINT;
	IM_TEN_MB_status : UDINT;
	IM_TEN_MB_inCommand_ARM : UINT;
	IM_SingleSignals_dP_maslo_gaz_Less100_status : UDINT;
	IM_SingleSignals_dp_kran1_Less100_status : UDINT;
	IM_SingleSignals_Razreshenie_zagruzki_dvig_status : UDINT;
	IM_SingleSignals_Vozbud_gotovnost_status : UDINT;
	IM_SingleSignals_Vozbud_neispr_tsepey_upr_AVR_pit_status : UDINT;
	IM_SingleSignals_Vozbud_neispravnost_status : UDINT;
	IM_SingleSignals_SHAVR1_v_rabote_status : UDINT;
	IM_SingleSignals_SHAVR2_v_rabote_status : UDINT;
	IM_SingleSignals_Avariinoe_otkluch_vikluchatelya_status : UDINT;
	IM_SingleSignals_Assinhronnii_hod_peregruzka_status : UDINT;
	IM_SingleSignals_SHU_v_GPA_vkluch_status : UDINT;
	IM_SingleSignals_SHP_v_GPA_vkluch_status : UDINT;
	IM_SingleSignals_QF1_on_status : UDINT;
	IM_SingleSignals_QF2_on_status : UDINT;
	IM_SingleSignals_QF23_on_status : UDINT;
	IM_SingleSignals_QF4_QF5_on_status : UDINT;
	IM_SingleSignals_QF6_QF7_on_status : UDINT;
	IM_SingleSignals_QF8_QF9_on_status : UDINT;
	IM_SingleSignals_QF10_QF11_on_status : UDINT;
	IM_SingleSignals_QF12_QF13_on_status : UDINT;
	IM_SingleSignals_QF14_QF15_on_status : UDINT;
	IM_SingleSignals_QF22_on_status : UDINT;
	IM_SingleSignals_NS_G1_G2_status : UDINT;
	IM_SingleSignals_NS_G3_G4_status : UDINT;
	IM_SingleSignals_NS_G15_G16_status : UDINT;
	IM_SingleSignals_NS_G17_status : UDINT;
	IM_SingleSignals_NS_G5_G6_status : UDINT;
	IM_SingleSignals_NS_G7_G8_status : UDINT;
	IM_SingleSignals_NS_G18_G19_status : UDINT;
	IM_SingleSignals_NS_G10_G11_status : UDINT;
	IM_SingleSignals_NS_G13_G14_status : UDINT;
	IM_SingleSignals_Uroven_masla_akkum_status : UDINT;
	IM_SingleSignals_NKU1_GPA_on_status : UDINT;
	IM_SingleSignals_NKU2_GPA_on_status : UDINT;
	IM_SingleSignals_AO_KC_ot_SHKS_status : UDINT;
	IM_SingleSignals_AO_GPA_ot_SHU_status : UDINT;
	IM_SingleSignals_BEAO_srabotal_status : UDINT;
	IM_SingleSignals_Chastotny_pusk_status : UDINT;
	IM_SingleSignals_Neuspesh_chastotny_pusk_status : UDINT;
	IM_SingleSignals_Rezhim_ruchnogo_regulirovaniya_status : UDINT;
	IM_SingleSignals_Osnovnoy_regul_off_status : UDINT;
	IM_SingleSignals_Voltage_sekcii_norm_status : UDINT;
	IM_SingleSignals_Reactorny_pusk_status : UDINT;
	IM_SingleSignals_NO_GPA_ot_SHU_status : UDINT;
	IM_SingleSignals_AO_GPA_ot_PRU_status : UDINT;
	IM_SingleSignals_Nalichie_BP1_status : UDINT;
	IM_SingleSignals_Nalichie_BP2_status : UDINT;
	IM_SingleSignals_Nalichie_BP3_status : UDINT;
	IM_SingleSignals_Nalichie_BP4_status : UDINT;
	IM_SingleSignals_Nalichie_BP5_status : UDINT;
	IM_SingleSignals_Nalichie_BP6_status : UDINT;
	IM_SingleSignals_Nalichie_BP7_BP8_status : UDINT;
	IM_SingleSignals_Nalichie_BP9_BP10_status : UDINT;
	IM_SingleSignals_Nalichie_cepei_upravlen_mv_status : UDINT;
	IM_SingleSignals_Nalichie_220BEAO_status : UDINT;
	IM_SingleSignals_Nalichie_per_220_na_vhode_status : UDINT;
	IM_SingleSignals_Nalichie_post_220_na_vhode_status : UDINT;
	IM_SingleSignals_Nalichie_BP11_status : UDINT;
	IM_SingleSignals_Nalichie_BP12_status : UDINT;
	IM_SingleSignals_Dver_SHU_pered_otkrita_status : UDINT;
	IM_SingleSignals_Dver_SHU_zad_otkrita_status : UDINT;
	IM_SingleSignals_EO_GPA_ot_knopki_SHU_status : UDINT;
	IM_SingleSignals_EO_EGPA_ot_PRY_status : UDINT;
	IM_SingleSignals_Synchroniz_rezhima_K1_status : UDINT;
	IM_SingleSignals_Potok_ms_posle_AVOM_status : UDINT;
END_VAR

IM_SingleSignals_dP_maslo_gaz_Less100_status := DWORD_TO_UDINT(Im.SingleSignals.dP_maslo_gaz_Less100.status);

IM_SingleSignals_dp_kran1_Less100_status := DWORD_TO_UDINT(Im.SingleSignals.dp_kran1_Less100.status);

IM_SingleSignals_Razreshenie_zagruzki_dvig_status := DWORD_TO_UDINT(Im.SingleSignals.Razreshenie_zagruzki_dvig.status);

IM_SingleSignals_Vozbud_gotovnost_status := DWORD_TO_UDINT(Im.SingleSignals.Vozbud_gotovnost.status);

IM_SingleSignals_Vozbud_neispr_tsepey_upr_AVR_pit_status := DWORD_TO_UDINT(Im.SingleSignals.Vozbud_neispr_tsepey_upr_AVR_pit.status);

IM_SingleSignals_Vozbud_neispravnost_status := DWORD_TO_UDINT(Im.SingleSignals.Vozbud_neispravnost.status);

IM_SingleSignals_SHAVR1_v_rabote_status := DWORD_TO_UDINT(Im.SingleSignals.SHAVR1_v_rabote.status);

IM_SingleSignals_SHAVR2_v_rabote_status := DWORD_TO_UDINT(Im.SingleSignals.SHAVR2_v_rabote.status);

IM_SingleSignals_Avariinoe_otkluch_vikluchatelya_status := DWORD_TO_UDINT(Im.SingleSignals.Avariinoe_otkluch_vikluchatelya.status);

IM_SingleSignals_Assinhronnii_hod_peregruzka_status := DWORD_TO_UDINT(Im.SingleSignals.Assinhronnii_hod_peregruzka.status);

IM_SingleSignals_SHU_v_GPA_vkluch_status := DWORD_TO_UDINT(Im.SingleSignals.SHU_v_GPA_vkluch.status);

IM_SingleSignals_SHP_v_GPA_vkluch_status := DWORD_TO_UDINT(Im.SingleSignals.SHP_v_GPA_vkluch.status);

IM_SingleSignals_QF1_on_status := DWORD_TO_UDINT(Im.SingleSignals.QF1_on.status);

IM_SingleSignals_QF2_on_status := DWORD_TO_UDINT(Im.SingleSignals.QF2_on.status);

IM_SingleSignals_QF23_on_status := DWORD_TO_UDINT(Im.SingleSignals.QF23_on.status);

IM_SingleSignals_QF4_QF5_on_status := DWORD_TO_UDINT(Im.SingleSignals.QF4_QF5_on.status);

IM_SingleSignals_QF6_QF7_on_status := DWORD_TO_UDINT(Im.SingleSignals.QF6_QF7_on.status);

IM_SingleSignals_QF8_QF9_on_status := DWORD_TO_UDINT(Im.SingleSignals.QF8_QF9_on.status);

IM_SingleSignals_QF10_QF11_on_status := DWORD_TO_UDINT(Im.SingleSignals.QF10_QF11_on.status);

IM_SingleSignals_QF12_QF13_on_status := DWORD_TO_UDINT(Im.SingleSignals.QF12_QF13_on.status);

IM_SingleSignals_QF14_QF15_on_status := DWORD_TO_UDINT(Im.SingleSignals.QF14_QF15_on.status);

IM_SingleSignals_QF22_on_status := DWORD_TO_UDINT(Im.SingleSignals.QF22_on.status);

IM_SingleSignals_NS_G1_G2_status := DWORD_TO_UDINT(Im.SingleSignals.NS_G1_G2.status);

IM_SingleSignals_NS_G3_G4_status := DWORD_TO_UDINT(Im.SingleSignals.NS_G3_G4.status);

IM_SingleSignals_NS_G15_G16_status := DWORD_TO_UDINT(Im.SingleSignals.NS_G15_G16.status);

IM_SingleSignals_NS_G17_status := DWORD_TO_UDINT(Im.SingleSignals.NS_G17.status);

IM_SingleSignals_NS_G5_G6_status := DWORD_TO_UDINT(Im.SingleSignals.NS_G5_G6.status);

IM_SingleSignals_NS_G7_G8_status := DWORD_TO_UDINT(Im.SingleSignals.NS_G7_G8.status);

IM_SingleSignals_NS_G18_G19_status := DWORD_TO_UDINT(Im.SingleSignals.NS_G18_G19.status);

IM_SingleSignals_NS_G10_G11_status := DWORD_TO_UDINT(Im.SingleSignals.NS_G10_G11.status);

IM_SingleSignals_NS_G13_G14_status := DWORD_TO_UDINT(Im.SingleSignals.NS_G13_G14.status);

IM_SingleSignals_Uroven_masla_akkum_status := DWORD_TO_UDINT(Im.SingleSignals.Uroven_masla_akkum.status);

IM_SingleSignals_NKU1_GPA_on_status := DWORD_TO_UDINT(Im.SingleSignals.NKU1_GPA_on.status);

IM_SingleSignals_NKU2_GPA_on_status := DWORD_TO_UDINT(Im.SingleSignals.NKU2_GPA_on.status);

IM_SingleSignals_AO_KC_ot_SHKS_status := DWORD_TO_UDINT(Im.SingleSignals.AO_KC_ot_SHKS.status);

IM_SingleSignals_AO_GPA_ot_SHU_status := DWORD_TO_UDINT(Im.SingleSignals.AO_GPA_ot_SHU.status);

IM_SingleSignals_BEAO_srabotal_status := DWORD_TO_UDINT(Im.SingleSignals.BEAO_srabotal.status);

IM_SingleSignals_Chastotny_pusk_status := DWORD_TO_UDINT(Im.SingleSignals.Chastotny_pusk.status);

IM_SingleSignals_Neuspesh_chastotny_pusk_status := DWORD_TO_UDINT(Im.SingleSignals.Neuspesh_chastotny_pusk.status);

IM_SingleSignals_Rezhim_ruchnogo_regulirovaniya_status := DWORD_TO_UDINT(Im.SingleSignals.Rezhim_ruchnogo_regulirovaniya.status);

IM_SingleSignals_Osnovnoy_regul_off_status := DWORD_TO_UDINT(Im.SingleSignals.Osnovnoy_regul_off.status);

IM_SingleSignals_Voltage_sekcii_norm_status := DWORD_TO_UDINT(Im.SingleSignals.Voltage_sekcii_norm.status);

IM_SingleSignals_Reactorny_pusk_status := DWORD_TO_UDINT(Im.SingleSignals.Reactorny_pusk.status);

IM_SingleSignals_NO_GPA_ot_SHU_status := DWORD_TO_UDINT(Im.SingleSignals.NO_GPA_ot_SHU.status);

IM_SingleSignals_AO_GPA_ot_PRU_status := DWORD_TO_UDINT(Im.SingleSignals.AO_GPA_ot_PRU.status);

IM_SingleSignals_Nalichie_BP1_status := DWORD_TO_UDINT(Im.SingleSignals.Nalichie_BP1.status);

IM_SingleSignals_Nalichie_BP2_status := DWORD_TO_UDINT(Im.SingleSignals.Nalichie_BP2.status);

IM_SingleSignals_Nalichie_BP3_status := DWORD_TO_UDINT(Im.SingleSignals.Nalichie_BP3.status);

IM_SingleSignals_Nalichie_BP4_status := DWORD_TO_UDINT(Im.SingleSignals.Nalichie_BP4.status);

IM_SingleSignals_Nalichie_BP5_status := DWORD_TO_UDINT(Im.SingleSignals.Nalichie_BP5.status);

IM_SingleSignals_Nalichie_BP6_status := DWORD_TO_UDINT(Im.SingleSignals.Nalichie_BP6.status);

IM_SingleSignals_Nalichie_BP7_BP8_status := DWORD_TO_UDINT(Im.SingleSignals.Nalichie_BP7_BP8.status);

IM_SingleSignals_Nalichie_BP9_BP10_status := DWORD_TO_UDINT(Im.SingleSignals.Nalichie_BP9_BP10.status);

IM_SingleSignals_Nalichie_cepei_upravlen_mv_status := DWORD_TO_UDINT(Im.SingleSignals.Nalichie_cepei_upravlen_mv.status);

IM_SingleSignals_Nalichie_220BEAO_status := DWORD_TO_UDINT(Im.SingleSignals.Nalichie_220BEAO.status);

IM_SingleSignals_Nalichie_per_220_na_vhode_status := DWORD_TO_UDINT(Im.SingleSignals.Nalichie_per_220_na_vhode.status);

IM_SingleSignals_Nalichie_post_220_na_vhode_status := DWORD_TO_UDINT(Im.SingleSignals.Nalichie_post_220_na_vhode.status);

IM_SingleSignals_Nalichie_BP11_status := DWORD_TO_UDINT(Im.SingleSignals.Nalichie_BP11.status);

IM_SingleSignals_Nalichie_BP12_status := DWORD_TO_UDINT(Im.SingleSignals.Nalichie_BP12.status);

IM_SingleSignals_Dver_SHU_pered_otkrita_status := DWORD_TO_UDINT(Im.SingleSignals.Dver_SHU_pered_otkrita.status);

IM_SingleSignals_Dver_SHU_zad_otkrita_status := DWORD_TO_UDINT(Im.SingleSignals.Dver_SHU_zad_otkrita.status);

IM_SingleSignals_EO_GPA_ot_knopki_SHU_status := DWORD_TO_UDINT(Im.SingleSignals.EO_GPA_ot_knopki_SHU.status);

IM_SingleSignals_EO_EGPA_ot_PRY_status := DWORD_TO_UDINT(Im.SingleSignals.EO_EGPA_ot_PRY.status);

IM_SingleSignals_Synchroniz_rezhima_K1_status := DWORD_TO_UDINT(Im.SingleSignals.Synchroniz_rezhima_K1.status);

IM_SingleSignals_Potok_ms_posle_AVOM_status := DWORD_TO_UDINT(Im.SingleSignals.Potok_ms_posle_AVOM.status);

IM_Kran1_status := DWORD_TO_UDINT(Im.Kran1.status);

IM_Kran2_status := DWORD_TO_UDINT(Im.Kran2.status);

IM_Kran3_status := DWORD_TO_UDINT(Im.Kran3.status);

IM_Kran3b_status := DWORD_TO_UDINT(Im.Kran3b.status);

IM_Kran4_status := DWORD_TO_UDINT(Im.Kran4.status);

IM_Kran5_status := DWORD_TO_UDINT(Im.Kran5.status);

IM_Kran6_status := DWORD_TO_UDINT(Im.Kran6.status);

IM_nu1_status := DWORD_TO_UDINT(Im.nu1.status);

IM_nu2_status := DWORD_TO_UDINT(Im.nu2.status);

IM_pns_status := DWORD_TO_UDINT(Im.pns.status);

IM_v1_Avom_status := DWORD_TO_UDINT(Im.v1_Avom.status);

IM_v2_Avom_status := DWORD_TO_UDINT(Im.v2_Avom.status);

IM_v3_Avom_status := DWORD_TO_UDINT(Im.v3_Avom.status);

IM_v4_Avom_status := DWORD_TO_UDINT(Im.v4_Avom.status);

IM_mv_status := DWORD_TO_UDINT(Im.mv.status);

IM_KaloriferAVOM_status := DWORD_TO_UDINT(Im.KaloriferAVOM.status);

IM_CMN_status := DWORD_TO_UDINT(Im.CMN.status);

IM_TEN_kollectora_status := DWORD_TO_UDINT(Im.TEN_kollectora.status);

IM_TEN_MB_status := DWORD_TO_UDINT(Im.TEN_MB.status);

(* ---- OPC_PROTECTIONS_GET.st ---- *)
FUNCTION_BLOCK OPC_PROTECTIONS_GET

VAR_EXTERNAL
	protections_Topornogo_podshipnika_EDT_1_inCommand_ARM : UINT;
	protections : ProtectionsConfig;
	protections_Topornogo_podshipnika_EDT_1_status : UDINT;
	protections_Toy_podshipnika_EDT_2_inCommand_ARM : UINT;
	protections_Toy_podshipnika_EDT_2_status : UDINT;
	protections_Toy_podshipnika_kol_EDT_3_inCommand_ARM : UINT;
	protections_Toy_podshipnika_kol_EDT_3_status : UDINT;
	protections_Toy_podshipnika_kol_EDT_4_inCommand_ARM : UINT;
	protections_Toy_podshipnika_kol_EDT_4_status : UDINT;
	protections_To_podshipnika_shest_red_EDT_5_inCommand_ARM : UINT;
	protections_To_podshipnika_shest_red_EDT_5_status : UDINT;
	protections_To_podshipnika_shest_red_EDT_6_inCommand_ARM : UINT;
	protections_To_podshipnika_shest_red_EDT_6_status : UDINT;
	protections_To_podshipnika_N_EDT_7_inCommand_ARM : UINT;
	protections_To_podshipnika_N_EDT_7_status : UDINT;
	protections_To_podshipnika_svob_konca_EDT_8_inCommand_ARM : UINT;
	protections_To_podshipnika_svob_konca_EDT_8_status : UDINT;
	protections_Ty_podshipnika_rab_kol_EDT_9_inCommand_ARM : UINT;
	protections_Ty_podshipnika_rab_kol_EDT_9_status : UDINT;
	protections_Typornogo_podshipnika_nerab_kolodok_HT_10_inCommand_ARM : UINT;
	protections_Typornogo_podshipnika_nerab_kolodok_HT_10_status : UDINT;
	protections_Tgaza_na_vyhode_H_inCommand_ARM : UINT;
	protections_Tgaza_na_vyhode_H_status : UDINT;
	protections_Os_sdvig_nagnetatelja_plus_inCommand_ARM : UINT;
	protections_Os_sdvig_nagnetatelja_plus_status : UDINT;
	protections_Os_sdvig_nagnetatelja_minus_inCommand_ARM : UINT;
	protections_Os_sdvig_nagnetatelja_minus_status : UDINT;
	protections_Pgaza_na_vyhode_nagnetatelia_GPA_STOP_inCommand_ARM : UINT;
	protections_Pgaza_na_vyhode_nagnetatelia_GPA_STOP_status : UDINT;
	protections_Pgaza_na_vhode_nagnetatelia_GPA_STOP_inCommand_ARM : UINT;
	protections_Pgaza_na_vhode_nagnetatelia_GPA_STOP_status : UDINT;
	protections_Pgaza_na_vyhode_nagnetatelia_inCommand_ARM : UINT;
	protections_Pgaza_na_vyhode_nagnetatelia_status : UDINT;
	protections_dPmaslo_gaz_inCommand_ARM : UINT;
	protections_dPmaslo_gaz_status : UDINT;
	protections_Pmaslo_sm_nizkoe_inCommand_ARM : UINT;
	protections_Pmaslo_sm_nizkoe_status : UDINT;
	protections_Pmaslo_sm_vysokoe_inCommand_ARM : UINT;
	protections_Pmaslo_sm_vysokoe_status : UDINT;
	protections_Vibro_skorost_OPED_T1_inCommand_ARM : UINT;
	protections_Vibro_skorost_OPED_T1_status : UDINT;
	protections_Vibro_skorost_OPED_T2_inCommand_ARM : UINT;
	protections_Vibro_skorost_OPED_T2_status : UDINT;
	protections_Vibro_skorost_OYP_kolesa_ED_T3_inCommand_ARM : UINT;
	protections_Vibro_skorost_OYP_kolesa_ED_T3_status : UDINT;
	protections_Vibro_skorost_OP_kolesa_RH_T4_inCommand_ARM : UINT;
	protections_Vibro_skorost_OP_kolesa_RH_T4_status : UDINT;
	protections_Vibro_skorost_OP_shesterni_RED_T5_inCommand_ARM : UINT;
	protections_Vibro_skorost_OP_shesterni_RED_T5_status : UDINT;
	protections_Vibro_skorost_OP_shesterni_RED_T6_inCommand_ARM : UINT;
	protections_Vibro_skorost_OP_shesterni_RED_T6_status : UDINT;
	protections_dPmaslo_gaz_less100_inCommand_ARM : UINT;
	protections_dPmaslo_gaz_less100_status : UDINT;
	protections_Reg_vozb_off_inCommand_ARM : UINT;
	protections_Reg_vozb_off_status : UDINT;
	protections_Fail_chastotnii_pusk_inCommand_ARM : UINT;
	protections_Fail_chastotnii_pusk_status : UDINT;
	protections_Off_avar_vikluchatel_inCommand_ARM : UINT;
	protections_Off_avar_vikluchatel_status : UDINT;
	protections_AOKC_SHKC_inCommand_ARM : UINT;
	protections_AOKC_SHKC_status : UDINT;
	protections_AO_PRU_inCommand_ARM : UINT;
	protections_AO_PRU_status : UDINT;
	protections_AO_ot_SHU_inCommand_ARM : UINT;
	protections_AO_ot_SHU_status : UDINT;
	protections_mvOff_inCommand_ARM : UINT;
	protections_mvOff_status : UDINT;
	protections_Kran1_sdvig_inCommand_ARM : UINT;
	protections_Kran1_sdvig_status : UDINT;
	protections_Kran2_sdvig_inCommand_ARM : UINT;
	protections_Kran2_sdvig_status : UDINT;
END_VAR

protections.Topornogo_podshipnika_EDT_1.inCommand_ARM := UINT_TO_WORD(protections_Topornogo_podshipnika_EDT_1_inCommand_ARM);

protections.Toy_podshipnika_EDT_2.inCommand_ARM := UINT_TO_WORD(protections_Toy_podshipnika_EDT_2_inCommand_ARM);

protections.Toy_podshipnika_kol_EDT_3.inCommand_ARM := UINT_TO_WORD(protections_Toy_podshipnika_kol_EDT_3_inCommand_ARM);

protections.Toy_podshipnika_kol_EDT_4.inCommand_ARM := UINT_TO_WORD(protections_Toy_podshipnika_kol_EDT_4_inCommand_ARM);

protections.To_podshipnika_shest_red_EDT_5.inCommand_ARM := UINT_TO_WORD(protections_To_podshipnika_shest_red_EDT_5_inCommand_ARM);

protections.To_podshipnika_shest_red_EDT_6.inCommand_ARM := UINT_TO_WORD(protections_To_podshipnika_shest_red_EDT_6_inCommand_ARM);

protections.To_podshipnika_N_EDT_7.inCommand_ARM := UINT_TO_WORD(protections_To_podshipnika_N_EDT_7_inCommand_ARM);

protections.To_podshipnika_svob_konca_EDT_8.inCommand_ARM := UINT_TO_WORD(protections_To_podshipnika_svob_konca_EDT_8_inCommand_ARM);

protections.Ty_podshipnika_rab_kol_EDT_9.inCommand_ARM := UINT_TO_WORD(protections_Ty_podshipnika_rab_kol_EDT_9_inCommand_ARM);

protections.Typornogo_podshipnika_nerab_kolodok_HT_10.inCommand_ARM := UINT_TO_WORD(protections_Typornogo_podshipnika_nerab_kolodok_HT_10_inCommand_ARM);

protections.Tgaza_na_vyhode_H.inCommand_ARM := UINT_TO_WORD(protections_Tgaza_na_vyhode_H_inCommand_ARM);

protections.Os_sdvig_nagnetatelja_plus.inCommand_ARM := UINT_TO_WORD(protections_Os_sdvig_nagnetatelja_plus_inCommand_ARM);

protections.Os_sdvig_nagnetatelja_minus.inCommand_ARM := UINT_TO_WORD(protections_Os_sdvig_nagnetatelja_minus_inCommand_ARM);

protections.Pgaza_na_vyhode_nagnetatelia_GPA_STOP.inCommand_ARM := UINT_TO_WORD(protections_Pgaza_na_vyhode_nagnetatelia_GPA_STOP_inCommand_ARM);

protections.Pgaza_na_vhode_nagnetatelia_GPA_STOP.inCommand_ARM := UINT_TO_WORD(protections_Pgaza_na_vhode_nagnetatelia_GPA_STOP_inCommand_ARM);

protections.Pgaza_na_vyhode_nagnetatelia.inCommand_ARM := UINT_TO_WORD(protections_Pgaza_na_vyhode_nagnetatelia_inCommand_ARM);

protections.dPmaslo_gaz.inCommand_ARM := UINT_TO_WORD(protections_dPmaslo_gaz_inCommand_ARM);

protections.Pmaslo_sm_nizkoe.inCommand_ARM := UINT_TO_WORD(protections_Pmaslo_sm_nizkoe_inCommand_ARM);

protections.Pmaslo_sm_vysokoe.inCommand_ARM := UINT_TO_WORD(protections_Pmaslo_sm_vysokoe_inCommand_ARM);

protections.Vibro_skorost_OPED_T1.inCommand_ARM := UINT_TO_WORD(protections_Vibro_skorost_OPED_T1_inCommand_ARM);

protections.Vibro_skorost_OPED_T2.inCommand_ARM := UINT_TO_WORD(protections_Vibro_skorost_OPED_T2_inCommand_ARM);

protections.Vibro_skorost_OYP_kolesa_ED_T3.inCommand_ARM := UINT_TO_WORD(protections_Vibro_skorost_OYP_kolesa_ED_T3_inCommand_ARM);

protections.Vibro_skorost_OP_kolesa_RH_T4.inCommand_ARM := UINT_TO_WORD(protections_Vibro_skorost_OP_kolesa_RH_T4_inCommand_ARM);

protections.Vibro_skorost_OP_shesterni_RED_T5.inCommand_ARM := UINT_TO_WORD(protections_Vibro_skorost_OP_shesterni_RED_T5_inCommand_ARM);

protections.Vibro_skorost_OP_shesterni_RED_T6.inCommand_ARM := UINT_TO_WORD(protections_Vibro_skorost_OP_shesterni_RED_T6_inCommand_ARM);

protections.dPmaslo_gaz_less100.inCommand_ARM := UINT_TO_WORD(protections_dPmaslo_gaz_less100_inCommand_ARM);

protections.Reg_vozb_off.inCommand_ARM := UINT_TO_WORD(protections_Reg_vozb_off_inCommand_ARM);

protections.Fail_chastotnii_pusk.inCommand_ARM := UINT_TO_WORD(protections_Fail_chastotnii_pusk_inCommand_ARM);

protections.Off_avar_vikluchatel.inCommand_ARM := UINT_TO_WORD(protections_Off_avar_vikluchatel_inCommand_ARM);

protections.AOKC_SHKC.inCommand_ARM := UINT_TO_WORD(protections_AOKC_SHKC_inCommand_ARM);

protections.AO_PRU.inCommand_ARM := UINT_TO_WORD(protections_AO_PRU_inCommand_ARM);

protections.AO_ot_SHU.inCommand_ARM := UINT_TO_WORD(protections_AO_ot_SHU_inCommand_ARM);

protections.mvOff.inCommand_ARM := UINT_TO_WORD(protections_mvOff_inCommand_ARM);

protections.Kran1_sdvig.inCommand_ARM := UINT_TO_WORD(protections_Kran1_sdvig_inCommand_ARM);

protections.Kran2_sdvig.inCommand_ARM := UINT_TO_WORD(protections_Kran2_sdvig_inCommand_ARM);

(* ---- OPC_PROTECTIONS_SET.st ---- *)
FUNCTION_BLOCK OPC_PROTECTIONS_SET

VAR_EXTERNAL
	protections : ProtectionsConfig;
	protections_Topornogo_podshipnika_EDT_1_inCommand_ARM : UINT;
	protections_Topornogo_podshipnika_EDT_1_status : UDINT;
	protections_Toy_podshipnika_EDT_2_inCommand_ARM : UINT;
	protections_Toy_podshipnika_EDT_2_status : UDINT;
	protections_Toy_podshipnika_kol_EDT_3_inCommand_ARM : UINT;
	protections_Toy_podshipnika_kol_EDT_3_status : UDINT;
	protections_Toy_podshipnika_kol_EDT_4_inCommand_ARM : UINT;
	protections_Toy_podshipnika_kol_EDT_4_status : UDINT;
	protections_To_podshipnika_shest_red_EDT_5_inCommand_ARM : UINT;
	protections_To_podshipnika_shest_red_EDT_5_status : UDINT;
	protections_To_podshipnika_shest_red_EDT_6_inCommand_ARM : UINT;
	protections_To_podshipnika_shest_red_EDT_6_status : UDINT;
	protections_To_podshipnika_N_EDT_7_inCommand_ARM : UINT;
	protections_To_podshipnika_N_EDT_7_status : UDINT;
	protections_To_podshipnika_svob_konca_EDT_8_inCommand_ARM : UINT;
	protections_To_podshipnika_svob_konca_EDT_8_status : UDINT;
	protections_Ty_podshipnika_rab_kol_EDT_9_inCommand_ARM : UINT;
	protections_Ty_podshipnika_rab_kol_EDT_9_status : UDINT;
	protections_Typornogo_podshipnika_nerab_kolodok_HT_10_inCommand_ARM : UINT;
	protections_Typornogo_podshipnika_nerab_kolodok_HT_10_status : UDINT;
	protections_Tgaza_na_vyhode_H_inCommand_ARM : UINT;
	protections_Tgaza_na_vyhode_H_status : UDINT;
	protections_Os_sdvig_nagnetatelja_plus_inCommand_ARM : UINT;
	protections_Os_sdvig_nagnetatelja_plus_status : UDINT;
	protections_Os_sdvig_nagnetatelja_minus_inCommand_ARM : UINT;
	protections_Os_sdvig_nagnetatelja_minus_status : UDINT;
	protections_Pgaza_na_vyhode_nagnetatelia_GPA_STOP_inCommand_ARM : UINT;
	protections_Pgaza_na_vyhode_nagnetatelia_GPA_STOP_status : UDINT;
	protections_Pgaza_na_vhode_nagnetatelia_GPA_STOP_inCommand_ARM : UINT;
	protections_Pgaza_na_vhode_nagnetatelia_GPA_STOP_status : UDINT;
	protections_Pgaza_na_vyhode_nagnetatelia_inCommand_ARM : UINT;
	protections_Pgaza_na_vyhode_nagnetatelia_status : UDINT;
	protections_dPmaslo_gaz_inCommand_ARM : UINT;
	protections_dPmaslo_gaz_status : UDINT;
	protections_Pmaslo_sm_nizkoe_inCommand_ARM : UINT;
	protections_Pmaslo_sm_nizkoe_status : UDINT;
	protections_Pmaslo_sm_vysokoe_inCommand_ARM : UINT;
	protections_Pmaslo_sm_vysokoe_status : UDINT;
	protections_Vibro_skorost_OPED_T1_inCommand_ARM : UINT;
	protections_Vibro_skorost_OPED_T1_status : UDINT;
	protections_Vibro_skorost_OPED_T2_inCommand_ARM : UINT;
	protections_Vibro_skorost_OPED_T2_status : UDINT;
	protections_Vibro_skorost_OYP_kolesa_ED_T3_inCommand_ARM : UINT;
	protections_Vibro_skorost_OYP_kolesa_ED_T3_status : UDINT;
	protections_Vibro_skorost_OP_kolesa_RH_T4_inCommand_ARM : UINT;
	protections_Vibro_skorost_OP_kolesa_RH_T4_status : UDINT;
	protections_Vibro_skorost_OP_shesterni_RED_T5_inCommand_ARM : UINT;
	protections_Vibro_skorost_OP_shesterni_RED_T5_status : UDINT;
	protections_Vibro_skorost_OP_shesterni_RED_T6_inCommand_ARM : UINT;
	protections_Vibro_skorost_OP_shesterni_RED_T6_status : UDINT;
	protections_dPmaslo_gaz_less100_inCommand_ARM : UINT;
	protections_dPmaslo_gaz_less100_status : UDINT;
	protections_Reg_vozb_off_inCommand_ARM : UINT;
	protections_Reg_vozb_off_status : UDINT;
	protections_Fail_chastotnii_pusk_inCommand_ARM : UINT;
	protections_Fail_chastotnii_pusk_status : UDINT;
	protections_Off_avar_vikluchatel_inCommand_ARM : UINT;
	protections_Off_avar_vikluchatel_status : UDINT;
	protections_AOKC_SHKC_inCommand_ARM : UINT;
	protections_AOKC_SHKC_status : UDINT;
	protections_AO_PRU_inCommand_ARM : UINT;
	protections_AO_PRU_status : UDINT;
	protections_AO_ot_SHU_inCommand_ARM : UINT;
	protections_AO_ot_SHU_status : UDINT;
	protections_mvOff_inCommand_ARM : UINT;
	protections_mvOff_status : UDINT;
	protections_Kran1_sdvig_inCommand_ARM : UINT;
	protections_Kran1_sdvig_status : UDINT;
	protections_Kran2_sdvig_inCommand_ARM : UINT;
	protections_Kran2_sdvig_status : UDINT;
END_VAR

    protections_Topornogo_podshipnika_EDT_1_status := DWORD_TO_UDINT(protections.Topornogo_podshipnika_EDT_1.status);

    protections_Toy_podshipnika_EDT_2_status := DWORD_TO_UDINT(protections.Toy_podshipnika_EDT_2.status);

    protections_Toy_podshipnika_kol_EDT_3_status := DWORD_TO_UDINT(protections.Toy_podshipnika_kol_EDT_3.status);

    protections_Toy_podshipnika_kol_EDT_4_status := DWORD_TO_UDINT(protections.Toy_podshipnika_kol_EDT_4.status);

    protections_To_podshipnika_shest_red_EDT_5_status := DWORD_TO_UDINT(protections.To_podshipnika_shest_red_EDT_5.status);

    protections_To_podshipnika_shest_red_EDT_6_status := DWORD_TO_UDINT(protections.To_podshipnika_shest_red_EDT_6.status);

    protections_To_podshipnika_N_EDT_7_status := DWORD_TO_UDINT(protections.To_podshipnika_N_EDT_7.status);

    protections_To_podshipnika_svob_konca_EDT_8_status := DWORD_TO_UDINT(protections.To_podshipnika_svob_konca_EDT_8.status);

    protections_Ty_podshipnika_rab_kol_EDT_9_status := DWORD_TO_UDINT(protections.Ty_podshipnika_rab_kol_EDT_9.status);

    protections_Typornogo_podshipnika_nerab_kolodok_HT_10_status := DWORD_TO_UDINT(protections.Typornogo_podshipnika_nerab_kolodok_HT_10.status);

    protections_Tgaza_na_vyhode_H_status := DWORD_TO_UDINT(protections.Tgaza_na_vyhode_H.status);

    protections_Os_sdvig_nagnetatelja_plus_status := DWORD_TO_UDINT(protections.Os_sdvig_nagnetatelja_plus.status);

    protections_Os_sdvig_nagnetatelja_minus_status := DWORD_TO_UDINT(protections.Os_sdvig_nagnetatelja_minus.status);

    protections_Pgaza_na_vyhode_nagnetatelia_GPA_STOP_status := DWORD_TO_UDINT(protections.Pgaza_na_vyhode_nagnetatelia_GPA_STOP.status);

    protections_Pgaza_na_vhode_nagnetatelia_GPA_STOP_status := DWORD_TO_UDINT(protections.Pgaza_na_vhode_nagnetatelia_GPA_STOP.status);

    protections_Pgaza_na_vyhode_nagnetatelia_status := DWORD_TO_UDINT(protections.Pgaza_na_vyhode_nagnetatelia.status);

    protections_dPmaslo_gaz_status := DWORD_TO_UDINT(protections.dPmaslo_gaz.status);

    protections_Pmaslo_sm_nizkoe_status := DWORD_TO_UDINT(protections.Pmaslo_sm_nizkoe.status);

    protections_Pmaslo_sm_vysokoe_status := DWORD_TO_UDINT(protections.Pmaslo_sm_vysokoe.status);

    protections_Vibro_skorost_OPED_T1_status := DWORD_TO_UDINT(protections.Vibro_skorost_OPED_T1.status);

    protections_Vibro_skorost_OPED_T2_status := DWORD_TO_UDINT(protections.Vibro_skorost_OPED_T2.status);

    protections_Vibro_skorost_OYP_kolesa_ED_T3_status := DWORD_TO_UDINT(protections.Vibro_skorost_OYP_kolesa_ED_T3.status);

    protections_Vibro_skorost_OP_kolesa_RH_T4_status := DWORD_TO_UDINT(protections.Vibro_skorost_OP_kolesa_RH_T4.status);

    protections_Vibro_skorost_OP_shesterni_RED_T5_status := DWORD_TO_UDINT(protections.Vibro_skorost_OP_shesterni_RED_T5.status);

    protections_Vibro_skorost_OP_shesterni_RED_T6_status := DWORD_TO_UDINT(protections.Vibro_skorost_OP_shesterni_RED_T6.status);

    protections_dPmaslo_gaz_less100_status := DWORD_TO_UDINT(protections.dPmaslo_gaz_less100.status);

    protections_Reg_vozb_off_status := DWORD_TO_UDINT(protections.Reg_vozb_off.status);

    protections_Fail_chastotnii_pusk_status := DWORD_TO_UDINT(protections.Fail_chastotnii_pusk.status);

    protections_Off_avar_vikluchatel_status := DWORD_TO_UDINT(protections.Off_avar_vikluchatel.status);

    protections_AOKC_SHKC_status := DWORD_TO_UDINT(protections.AOKC_SHKC.status);

    protections_AO_PRU_status := DWORD_TO_UDINT(protections.AO_PRU.status);

    protections_AO_ot_SHU_status := DWORD_TO_UDINT(protections.AO_ot_SHU.status);

    protections_mvOff_status := DWORD_TO_UDINT(protections.mvOff.status);

    protections_Kran1_sdvig_status := DWORD_TO_UDINT(protections.Kran1_sdvig.status);

    protections_Kran2_sdvig_status := DWORD_TO_UDINT(protections.Kran2_sdvig.status);

(* ---- ph_SingleOutput.st ---- *)
FUNCTION_BLOCK ph_SingleOutput

VAR_IN_OUT
	im : struct_singleOutput;
END_VAR

VAR_INPUT
	WhatCanIdo : BOOL;
	PhaseNumber : UINT;
END_VAR

VAR_IN_OUT
	StrPh : struct_PhaseAlgoritm;
END_VAR

VAR
	reset_Trig : R_TRIG;
END_VAR

IF StrPh.run AND NOT StrPh.start THEN
	StrPh.start := TRUE;
	StrPh.top := FALSE;
	StrPh.error := FALSE;
          StrPh.run:=FALSE;

	IF (WhatCanIdo) THEN
	runIfNotRunningSO(im);
          ELSE
	resetIfRunningSO(im);
          END_IF;
END_IF;

IF StrPh.start AND NOT StrPh.top THEN
StrPh.top := (im.Q = WhatCanIdo);
END_IF;

reset_Trig(CLK := StrPh.reset);
IF reset_Trig.Q THEN
	StrPh.start := FALSE;
	StrPh.error := FALSE;
	StrPh.top := FALSE;
          StrPh.run:=FALSE;
          StrPh.reset:=FALSE;
END_IF;

StrPh.startStatus := SHL(BOOL_TO_DWORD(StrPh.start), PhaseNumber);
StrPh.errorStatus := SHL(BOOL_TO_DWORD(StrPh.error), PhaseNumber);
StrPh.topStatus := SHL(BOOL_TO_DWORD(StrPh.top), PhaseNumber);

(* ---- ph_SingleSignal.st ---- *)
FUNCTION_BLOCK ph_SingleSignal

VAR_IN_OUT
	im : struct_singleSignal;
END_VAR

VAR_INPUT
	expectedValue : BOOL          := TRUE;
	PhaseNumber : UINT;
END_VAR

VAR_IN_OUT
	StrPh : struct_PhaseAlgoritm;
END_VAR

VAR
	reset_Trig : R_TRIG;
END_VAR

IF StrPh.run AND NOT StrPh.start THEN
	StrPh.start := TRUE;
	StrPh.top := FALSE;
	StrPh.error := FALSE;
          StrPh.run:=FALSE;
END_IF;

IF StrPh.start AND NOT StrPh.top THEN
StrPh.error:= NOT Im.reliability;
StrPh.top := (Im.Q = expectedValue) AND (Im.reliability);
END_IF;

reset_Trig(CLK := StrPh.reset);
IF reset_Trig.Q THEN
	StrPh.start := FALSE;
	StrPh.error := FALSE;
	StrPh.top := FALSE;
          StrPh.run:=FALSE;
          StrPh.reset:=FALSE;
END_IF;

StrPh.startStatus := SHL(BOOL_TO_DWORD(StrPh.start), PhaseNumber);
StrPh.errorStatus := SHL(BOOL_TO_DWORD(StrPh.error), PhaseNumber);
StrPh.topStatus := SHL(BOOL_TO_DWORD(StrPh.top), PhaseNumber);
